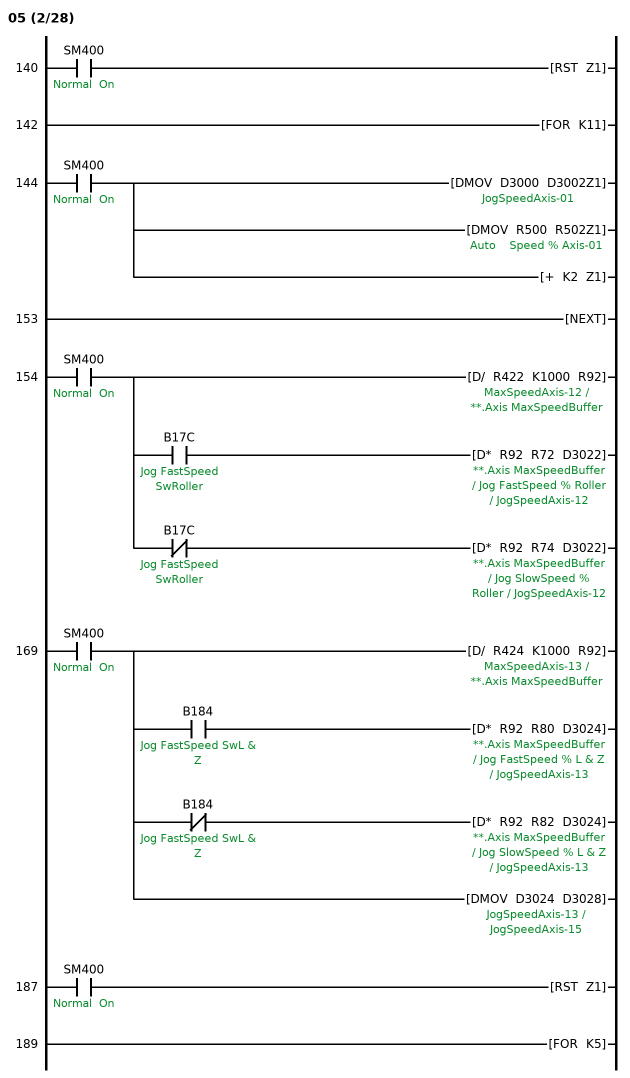
140   LD      SM400  ; Normal  On
      RST     Z1
142   FOR     K11
144   LD      SM400  ; Normal  On
      DMOV    D3000 D3002Z1
      DMOV    R500 R502Z1  ; Auto    Speed % Axis-01
      +       K2 Z1
153   NEXT
154   LD      SM400  ; Normal  On
      D/      R422 K1000 R92
      MPS
      AND     B17C  ; Jog FastSpeed SwRoller
      D*      R92 R72 D3022  ; Jog FastSpeed % Roller / JogSpeedAxis-12
      MPP
      ANI     B17C  ; Jog FastSpeed SwRoller
      D*      R92 R74 D3022  ; Jog SlowSpeed % Roller
169   LD      SM400  ; Normal  On
      D/      R424 K1000 R92
      MPS
      AND     B184  ; Jog FastSpeed SwL & Z
      D*      R92 R80 D3024  ; Jog FastSpeed % L & Z / JogSpeedAxis-13
      MRD
      ANI     B184  ; Jog FastSpeed SwL & Z
      D*      R92 R82 D3024  ; Jog SlowSpeed % L & Z
      MPP
      DMOV    D3024 D3028  ; JogSpeedAxis-15
187   LD      SM400  ; Normal  On
      RST     Z1
189   FOR     K5
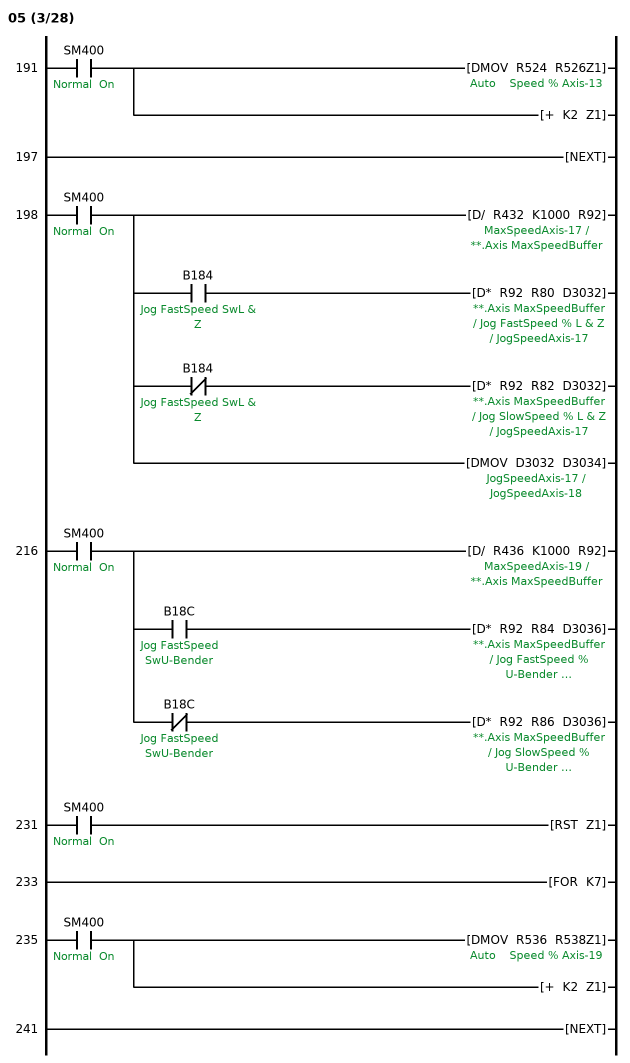
191   LD      SM400  ; Normal  On
      DMOV    R524 R526Z1  ; Auto    Speed % Axis-13
      +       K2 Z1
197   NEXT
198   LD      SM400  ; Normal  On
      D/      R432 K1000 R92  ; MaxSpeedAxis-17
      MPS
      AND     B184  ; Jog FastSpeed SwL & Z
      D*      R92 R80 D3032  ; JogSpeedAxis-17
      MRD
      ANI     B184  ; Jog FastSpeed SwL & Z
      D*      R92 R82 D3032
      MPP
      DMOV    D3032 D3034  ; JogSpeedAxis-18
216   LD      SM400  ; Normal  On
      D/      R436 K1000 R92
      MPS
      AND     B18C  ; Jog FastSpeed SwU-Bender
      D*      R92 R84 D3036  ; Jog FastSpeed % U-Bender / JogSpeedAxis-19
      MPP
      ANI     B18C  ; Jog FastSpeed SwU-Bender
      D*      R92 R86 D3036  ; Jog SlowSpeed % U-Bender
231   LD      SM400  ; Normal  On
      RST     Z1
233   FOR     K7
235   LD      SM400  ; Normal  On
      DMOV    R536 R538Z1  ; Auto    Speed % Axis-19
      +       K2 Z1
241   NEXT
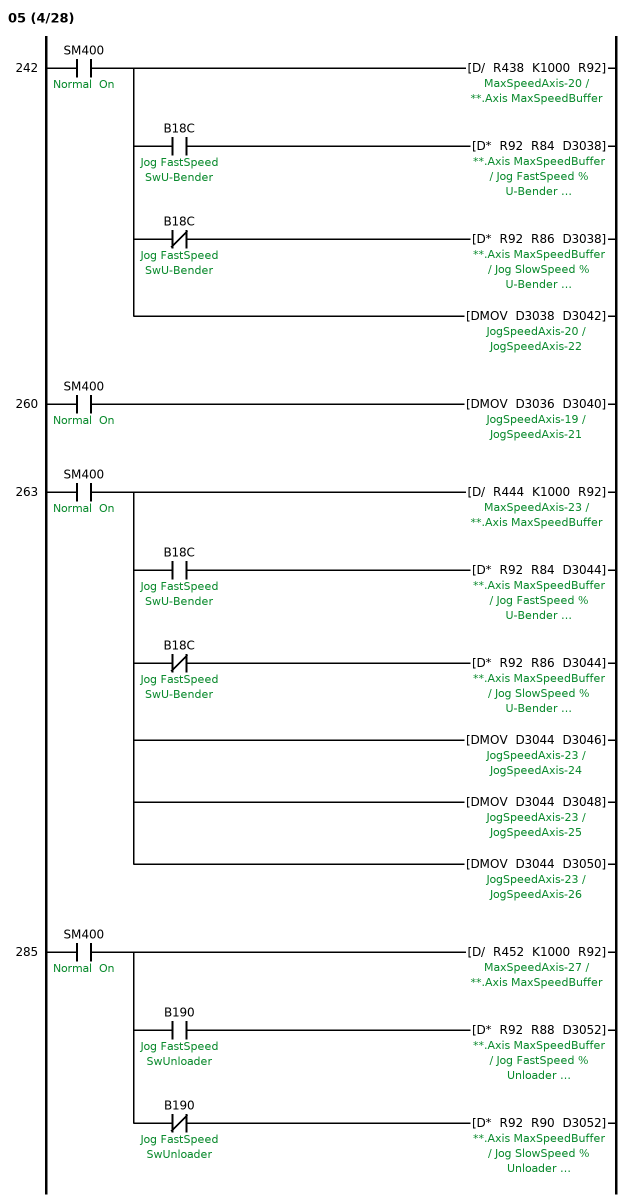
242   LD      SM400  ; Normal  On
      D/      R438 K1000 R92
      MPS
      AND     B18C  ; Jog FastSpeed SwU-Bender
      D*      R92 R84 D3038  ; JogSpeedAxis-20
      MRD
      ANI     B18C  ; Jog FastSpeed SwU-Bender
      D*      R92 R86 D3038
      MPP
      DMOV    D3038 D3042  ; JogSpeedAxis-22
260   LD      SM400  ; Normal  On
      DMOV    D3036 D3040  ; JogSpeedAxis-21
263   LD      SM400  ; Normal  On
      D/      R444 K1000 R92  ; MaxSpeedAxis-23
      MPS
      AND     B18C  ; Jog FastSpeed SwU-Bender
      D*      R92 R84 D3044  ; JogSpeedAxis-23
      MRD
      ANI     B18C  ; Jog FastSpeed SwU-Bender
      D*      R92 R86 D3044
      MPP
      DMOV    D3044 D3046  ; JogSpeedAxis-24
      DMOV    D3044 D3048  ; JogSpeedAxis-25
      DMOV    D3044 D3050  ; JogSpeedAxis-26
285   LD      SM400  ; Normal  On
      D/      R452 K1000 R92
      MPS
      AND     B190  ; Jog FastSpeed SwUnloader
      D*      R92 R88 D3052  ; Jog FastSpeed % Unloader / JogSpeedAxis-27
      MPP
      ANI     B190  ; Jog FastSpeed SwUnloader
      D*      R92 R90 D3052  ; Jog SlowSpeed % Unloader
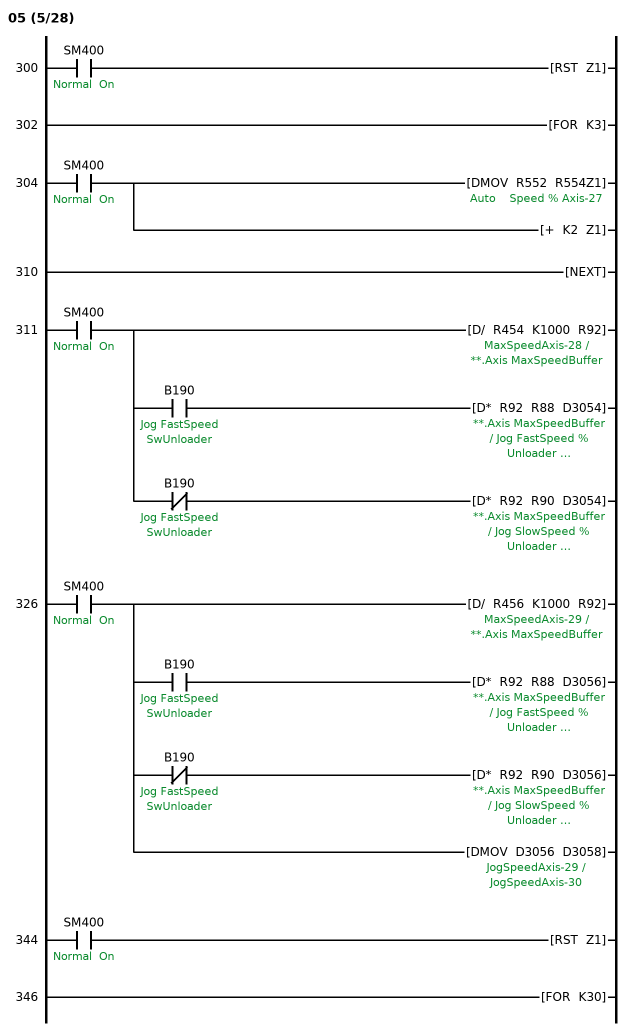
300   LD      SM400  ; Normal  On
      RST     Z1
302   FOR     K3
304   LD      SM400  ; Normal  On
      DMOV    R552 R554Z1  ; Auto    Speed % Axis-27
      +       K2 Z1
310   NEXT
311   LD      SM400  ; Normal  On
      D/      R454 K1000 R92
      MPS
      AND     B190  ; Jog FastSpeed SwUnloader
      D*      R92 R88 D3054  ; JogSpeedAxis-28
      MPP
      ANI     B190  ; Jog FastSpeed SwUnloader
      D*      R92 R90 D3054
326   LD      SM400  ; Normal  On
      D/      R456 K1000 R92  ; MaxSpeedAxis-29
      MPS
      AND     B190  ; Jog FastSpeed SwUnloader
      D*      R92 R88 D3056  ; JogSpeedAxis-29
      MRD
      ANI     B190  ; Jog FastSpeed SwUnloader
      D*      R92 R90 D3056
      MPP
      DMOV    D3056 D3058  ; JogSpeedAxis-30
344   LD      SM400  ; Normal  On
      RST     Z1
346   FOR     K30
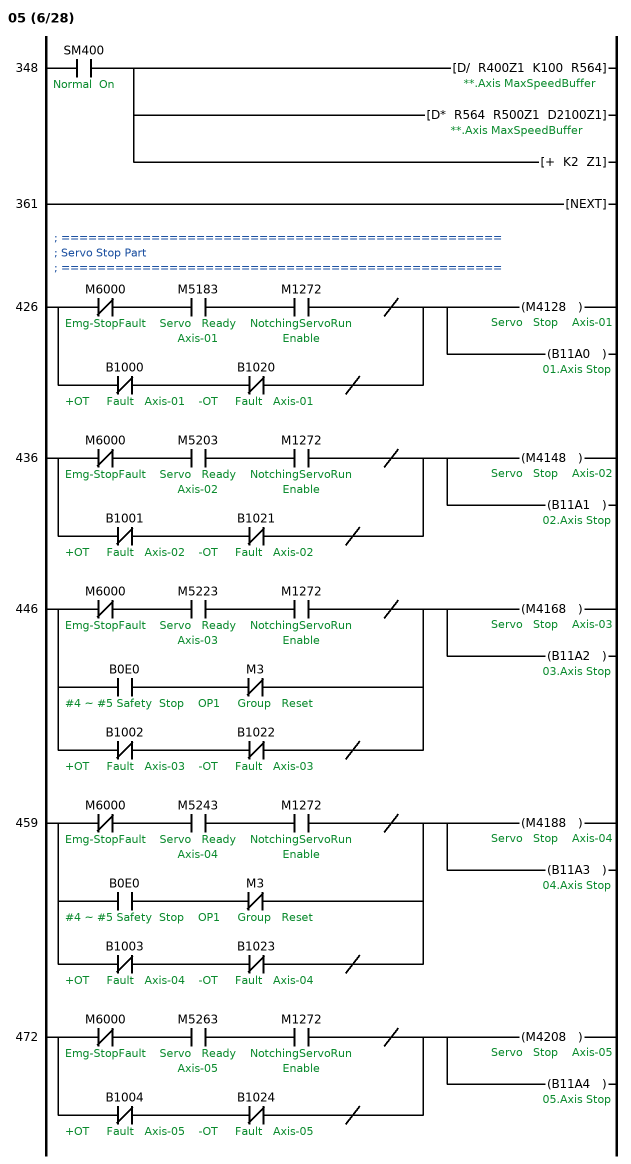
348   LD      SM400  ; Normal  On
      D/      R400Z1 K100 R564  ; **.Axis MaxSpeedBuffer
      D*      R564 R500Z1 D2100Z1
      +       K2 Z1
361   NEXT
; =================================================
; Servo Stop Part
; =================================================
426   LDI     M6000  ; Emg-StopFault
      AND     M5183  ; Servo   Ready   Axis-01
      AND     M1272  ; NotchingServoRunEnable
      INV
      LDI     B1000  ; +OT     Fault   Axis-01
      ANI     B1020  ; -OT     Fault   Axis-01
      INV
      ORB
      OUT     M4128  ; Servo   Stop    Axis-01
      OUT     B11A0  ; 01.Axis Stop
436   LDI     M6000  ; Emg-StopFault
      AND     M5203  ; Servo   Ready   Axis-02
      AND     M1272  ; NotchingServoRunEnable
      INV
      LDI     B1001  ; +OT     Fault   Axis-02
      ANI     B1021  ; -OT     Fault   Axis-02
      INV
      ORB
      OUT     M4148  ; Servo   Stop    Axis-02
      OUT     B11A1  ; 02.Axis Stop
446   LDI     M6000  ; Emg-StopFault
      AND     M5223  ; Servo   Ready   Axis-03
      AND     M1272  ; NotchingServoRunEnable
      INV
      LD      B0E0  ; #4 ~ #5 Safety  Stop
      ANI     M3  ; OP1     Group   Reset
      ORB
      LDI     B1002  ; +OT     Fault   Axis-03
      ANI     B1022  ; -OT     Fault   Axis-03
      INV
      ORB
      OUT     M4168  ; Servo   Stop    Axis-03
      OUT     B11A2  ; 03.Axis Stop
459   LDI     M6000  ; Emg-StopFault
      AND     M5243  ; Servo   Ready   Axis-04
      AND     M1272  ; NotchingServoRunEnable
      INV
      LD      B0E0  ; #4 ~ #5 Safety  Stop
      ANI     M3  ; OP1     Group   Reset
      ORB
      LDI     B1003  ; +OT     Fault   Axis-04
      ANI     B1023  ; -OT     Fault   Axis-04
      INV
      ORB
      OUT     M4188  ; Servo   Stop    Axis-04
      OUT     B11A3  ; 04.Axis Stop
472   LDI     M6000  ; Emg-StopFault
      AND     M5263  ; Servo   Ready   Axis-05
      AND     M1272  ; NotchingServoRunEnable
      INV
      LDI     B1004  ; +OT     Fault   Axis-05
      ANI     B1024  ; -OT     Fault   Axis-05
      INV
      ORB
      OUT     M4208  ; Servo   Stop    Axis-05
      OUT     B11A4  ; 05.Axis Stop
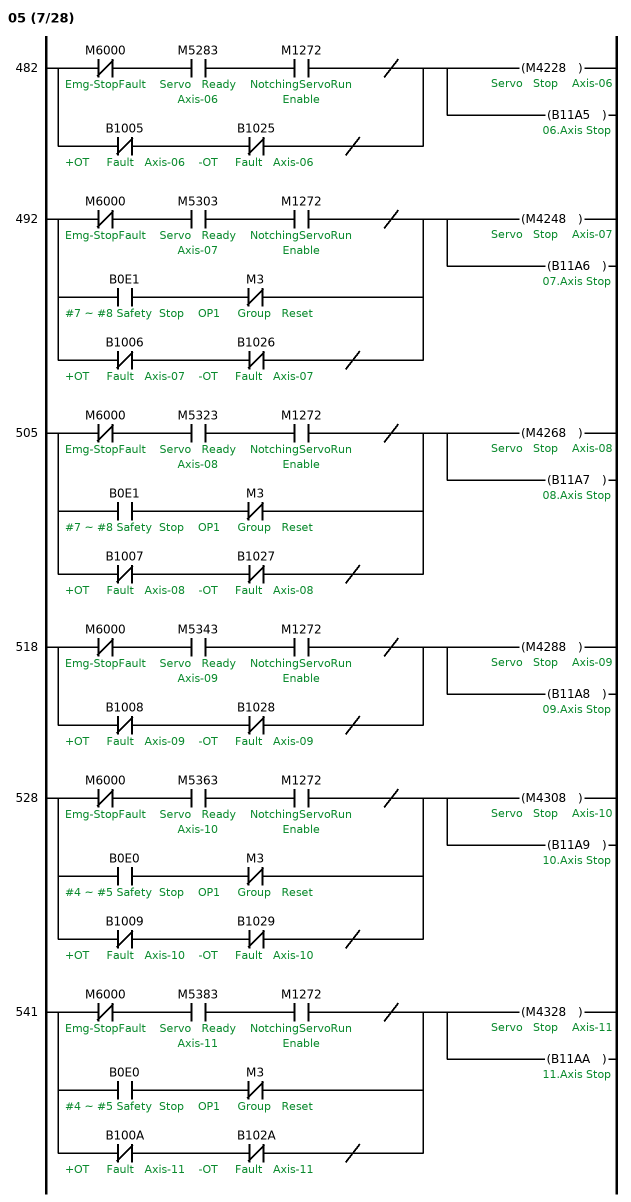
482   LDI     M6000  ; Emg-StopFault
      AND     M5283  ; Servo   Ready   Axis-06
      AND     M1272  ; NotchingServoRunEnable
      INV
      LDI     B1005  ; +OT     Fault   Axis-06
      ANI     B1025  ; -OT     Fault   Axis-06
      INV
      ORB
      OUT     M4228  ; Servo   Stop    Axis-06
      OUT     B11A5  ; 06.Axis Stop
492   LDI     M6000  ; Emg-StopFault
      AND     M5303  ; Servo   Ready   Axis-07
      AND     M1272  ; NotchingServoRunEnable
      INV
      LD      B0E1  ; #7 ~ #8 Safety  Stop
      ANI     M3  ; OP1     Group   Reset
      ORB
      LDI     B1006  ; +OT     Fault   Axis-07
      ANI     B1026  ; -OT     Fault   Axis-07
      INV
      ORB
      OUT     M4248  ; Servo   Stop    Axis-07
      OUT     B11A6  ; 07.Axis Stop
505   LDI     M6000  ; Emg-StopFault
      AND     M5323  ; Servo   Ready   Axis-08
      AND     M1272  ; NotchingServoRunEnable
      INV
      LD      B0E1  ; #7 ~ #8 Safety  Stop
      ANI     M3  ; OP1     Group   Reset
      ORB
      LDI     B1007  ; +OT     Fault   Axis-08
      ANI     B1027  ; -OT     Fault   Axis-08
      INV
      ORB
      OUT     M4268  ; Servo   Stop    Axis-08
      OUT     B11A7  ; 08.Axis Stop
518   LDI     M6000  ; Emg-StopFault
      AND     M5343  ; Servo   Ready   Axis-09
      AND     M1272  ; NotchingServoRunEnable
      INV
      LDI     B1008  ; +OT     Fault   Axis-09
      ANI     B1028  ; -OT     Fault   Axis-09
      INV
      ORB
      OUT     M4288  ; Servo   Stop    Axis-09
      OUT     B11A8  ; 09.Axis Stop
528   LDI     M6000  ; Emg-StopFault
      AND     M5363  ; Servo   Ready   Axis-10
      AND     M1272  ; NotchingServoRunEnable
      INV
      LD      B0E0  ; #4 ~ #5 Safety  Stop
      ANI     M3  ; OP1     Group   Reset
      ORB
      LDI     B1009  ; +OT     Fault   Axis-10
      ANI     B1029  ; -OT     Fault   Axis-10
      INV
      ORB
      OUT     M4308  ; Servo   Stop    Axis-10
      OUT     B11A9  ; 10.Axis Stop
541   LDI     M6000  ; Emg-StopFault
      AND     M5383  ; Servo   Ready   Axis-11
      AND     M1272  ; NotchingServoRunEnable
      INV
      LD      B0E0  ; #4 ~ #5 Safety  Stop
      ANI     M3  ; OP1     Group   Reset
      ORB
      LDI     B100A  ; +OT     Fault   Axis-11
      ANI     B102A  ; -OT     Fault   Axis-11
      INV
      ORB
      OUT     M4328  ; Servo   Stop    Axis-11
      OUT     B11AA  ; 11.Axis Stop
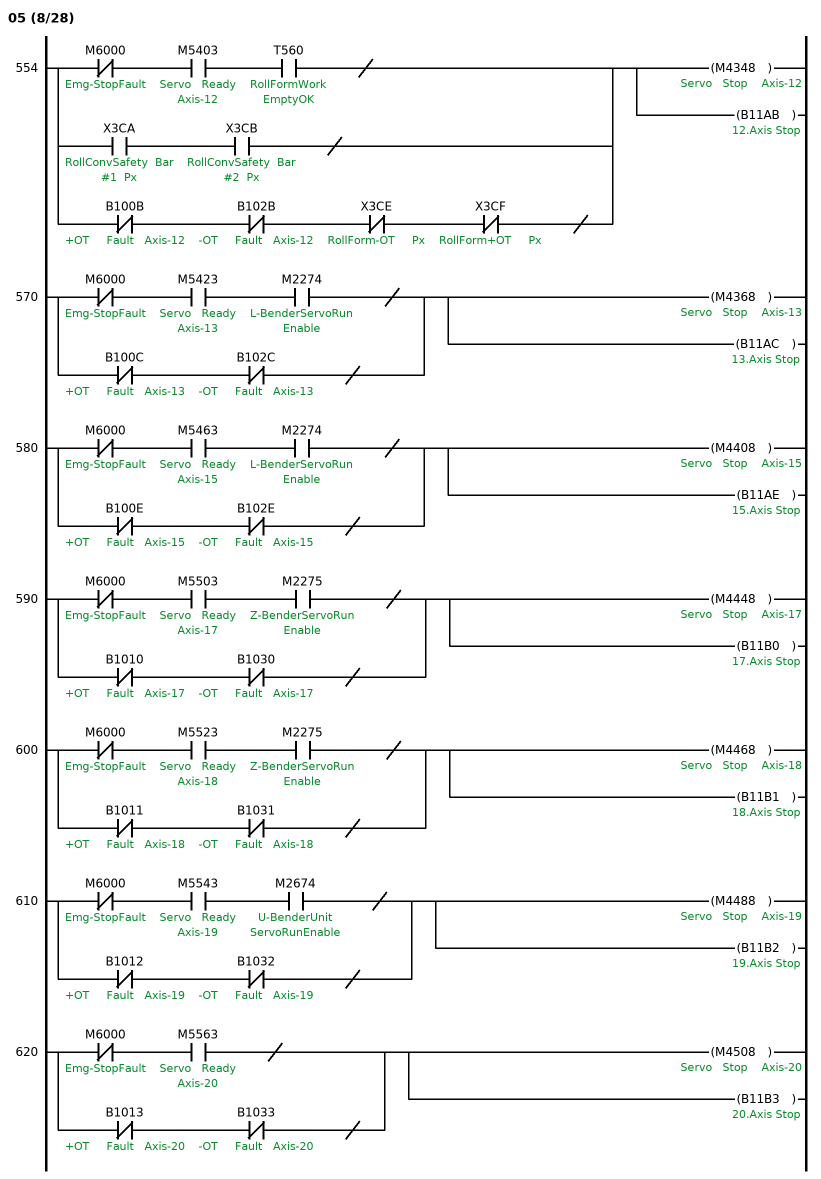
554   LDI     M6000  ; Emg-StopFault
      AND     M5403  ; Servo   Ready   Axis-12
      AND     T560  ; RollFormWork    EmptyOK
      INV
      LD      X3CA  ; RollConvSafety  Bar #1  Px
      AND     X3CB  ; RollConvSafety  Bar #2  Px
      INV
      ORB
      LDI     B100B  ; +OT     Fault   Axis-12
      ANI     B102B  ; -OT     Fault   Axis-12
      ANI     X3CE  ; RollForm-OT     Px
      ANI     X3CF  ; RollForm+OT     Px
      INV
      ORB
      OUT     M4348  ; Servo   Stop    Axis-12
      OUT     B11AB  ; 12.Axis Stop
570   LDI     M6000  ; Emg-StopFault
      AND     M5423  ; Servo   Ready   Axis-13
      AND     M2274  ; L-BenderServoRunEnable
      INV
      LDI     B100C  ; +OT     Fault   Axis-13
      ANI     B102C  ; -OT     Fault   Axis-13
      INV
      ORB
      OUT     M4368  ; Servo   Stop    Axis-13
      OUT     B11AC  ; 13.Axis Stop
580   LDI     M6000  ; Emg-StopFault
      AND     M5463  ; Servo   Ready   Axis-15
      AND     M2274  ; L-BenderServoRunEnable
      INV
      LDI     B100E  ; +OT     Fault   Axis-15
      ANI     B102E  ; -OT     Fault   Axis-15
      INV
      ORB
      OUT     M4408  ; Servo   Stop    Axis-15
      OUT     B11AE  ; 15.Axis Stop
590   LDI     M6000  ; Emg-StopFault
      AND     M5503  ; Servo   Ready   Axis-17
      AND     M2275  ; Z-BenderServoRunEnable
      INV
      LDI     B1010  ; +OT     Fault   Axis-17
      ANI     B1030  ; -OT     Fault   Axis-17
      INV
      ORB
      OUT     M4448  ; Servo   Stop    Axis-17
      OUT     B11B0  ; 17.Axis Stop
600   LDI     M6000  ; Emg-StopFault
      AND     M5523  ; Servo   Ready   Axis-18
      AND     M2275  ; Z-BenderServoRunEnable
      INV
      LDI     B1011  ; +OT     Fault   Axis-18
      ANI     B1031  ; -OT     Fault   Axis-18
      INV
      ORB
      OUT     M4468  ; Servo   Stop    Axis-18
      OUT     B11B1  ; 18.Axis Stop
610   LDI     M6000  ; Emg-StopFault
      AND     M5543  ; Servo   Ready   Axis-19
      AND     M2674  ; U-BenderUnit    ServoRunEnable
      INV
      LDI     B1012  ; +OT     Fault   Axis-19
      ANI     B1032  ; -OT     Fault   Axis-19
      INV
      ORB
      OUT     M4488  ; Servo   Stop    Axis-19
      OUT     B11B2  ; 19.Axis Stop
620   LDI     M6000  ; Emg-StopFault
      AND     M5563  ; Servo   Ready   Axis-20
      INV
      LDI     B1013  ; +OT     Fault   Axis-20
      ANI     B1033  ; -OT     Fault   Axis-20
      INV
      ORB
      OUT     M4508  ; Servo   Stop    Axis-20
      OUT     B11B3  ; 20.Axis Stop
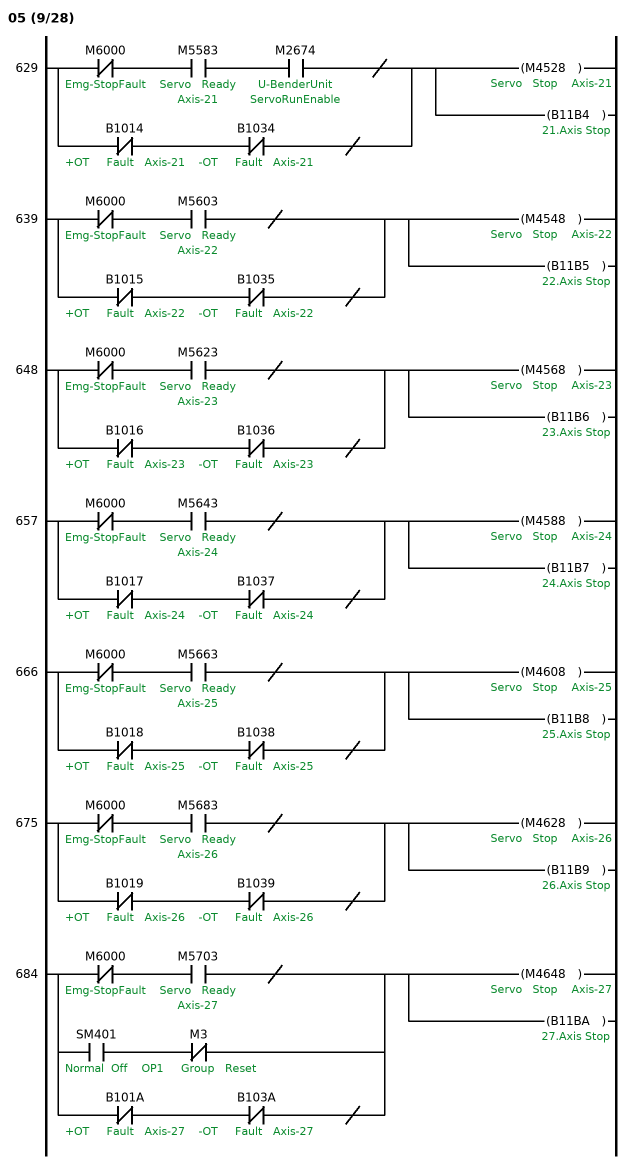
629   LDI     M6000  ; Emg-StopFault
      AND     M5583  ; Servo   Ready   Axis-21
      AND     M2674  ; U-BenderUnit    ServoRunEnable
      INV
      LDI     B1014  ; +OT     Fault   Axis-21
      ANI     B1034  ; -OT     Fault   Axis-21
      INV
      ORB
      OUT     M4528  ; Servo   Stop    Axis-21
      OUT     B11B4  ; 21.Axis Stop
639   LDI     M6000  ; Emg-StopFault
      AND     M5603  ; Servo   Ready   Axis-22
      INV
      LDI     B1015  ; +OT     Fault   Axis-22
      ANI     B1035  ; -OT     Fault   Axis-22
      INV
      ORB
      OUT     M4548  ; Servo   Stop    Axis-22
      OUT     B11B5  ; 22.Axis Stop
648   LDI     M6000  ; Emg-StopFault
      AND     M5623  ; Servo   Ready   Axis-23
      INV
      LDI     B1016  ; +OT     Fault   Axis-23
      ANI     B1036  ; -OT     Fault   Axis-23
      INV
      ORB
      OUT     M4568  ; Servo   Stop    Axis-23
      OUT     B11B6  ; 23.Axis Stop
657   LDI     M6000  ; Emg-StopFault
      AND     M5643  ; Servo   Ready   Axis-24
      INV
      LDI     B1017  ; +OT     Fault   Axis-24
      ANI     B1037  ; -OT     Fault   Axis-24
      INV
      ORB
      OUT     M4588  ; Servo   Stop    Axis-24
      OUT     B11B7  ; 24.Axis Stop
666   LDI     M6000  ; Emg-StopFault
      AND     M5663  ; Servo   Ready   Axis-25
      INV
      LDI     B1018  ; +OT     Fault   Axis-25
      ANI     B1038  ; -OT     Fault   Axis-25
      INV
      ORB
      OUT     M4608  ; Servo   Stop    Axis-25
      OUT     B11B8  ; 25.Axis Stop
675   LDI     M6000  ; Emg-StopFault
      AND     M5683  ; Servo   Ready   Axis-26
      INV
      LDI     B1019  ; +OT     Fault   Axis-26
      ANI     B1039  ; -OT     Fault   Axis-26
      INV
      ORB
      OUT     M4628  ; Servo   Stop    Axis-26
      OUT     B11B9  ; 26.Axis Stop
684   LDI     M6000  ; Emg-StopFault
      AND     M5703  ; Servo   Ready   Axis-27
      INV
      LD      SM401  ; Normal  Off
      ANI     M3  ; OP1     Group   Reset
      ORB
      LDI     B101A  ; +OT     Fault   Axis-27
      ANI     B103A  ; -OT     Fault   Axis-27
      INV
      ORB
      OUT     M4648  ; Servo   Stop    Axis-27
      OUT     B11BA  ; 27.Axis Stop
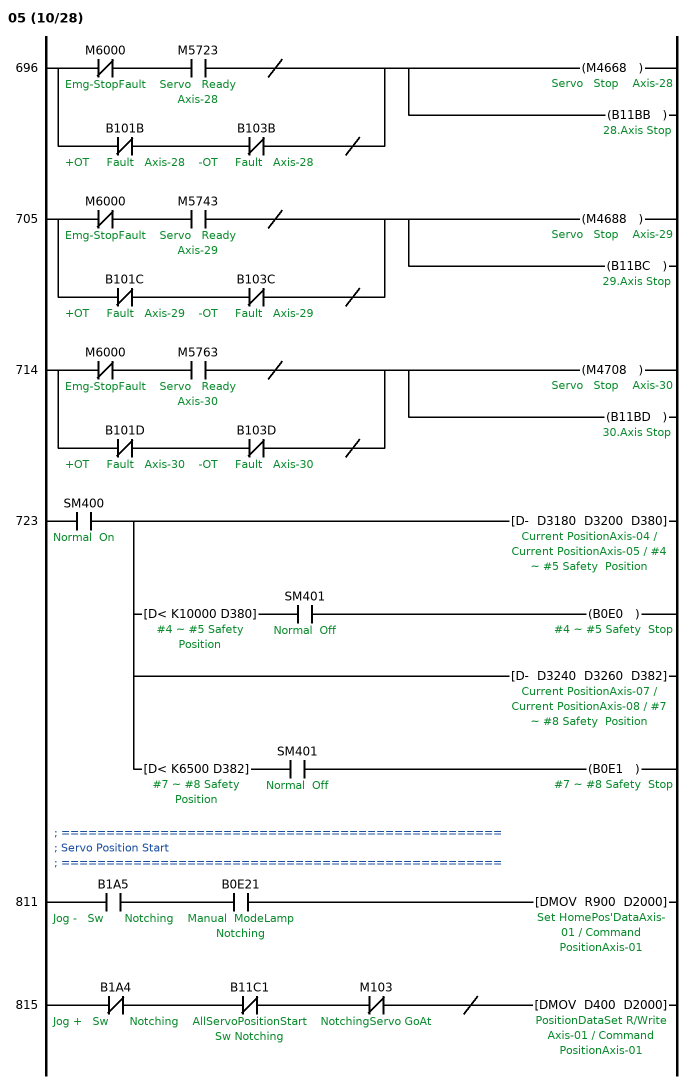
696   LDI     M6000  ; Emg-StopFault
      AND     M5723  ; Servo   Ready   Axis-28
      INV
      LDI     B101B  ; +OT     Fault   Axis-28
      ANI     B103B  ; -OT     Fault   Axis-28
      INV
      ORB
      OUT     M4668  ; Servo   Stop    Axis-28
      OUT     B11BB  ; 28.Axis Stop
705   LDI     M6000  ; Emg-StopFault
      AND     M5743  ; Servo   Ready   Axis-29
      INV
      LDI     B101C  ; +OT     Fault   Axis-29
      ANI     B103C  ; -OT     Fault   Axis-29
      INV
      ORB
      OUT     M4688  ; Servo   Stop    Axis-29
      OUT     B11BC  ; 29.Axis Stop
714   LDI     M6000  ; Emg-StopFault
      AND     M5763  ; Servo   Ready   Axis-30
      INV
      LDI     B101D  ; +OT     Fault   Axis-30
      ANI     B103D  ; -OT     Fault   Axis-30
      INV
      ORB
      OUT     M4708  ; Servo   Stop    Axis-30
      OUT     B11BD  ; 30.Axis Stop
723   LD      SM400  ; Normal  On
      D-      D3180 D3200 D380  ; Current PositionAxis-04 / Current PositionAxis-05 / #4 ~ #5 Safety  Position
      MPS
      ANDD<   K10000 D380  ; #4 ~ #5 Safety  Position
      AND     SM401  ; Normal  Off
      OUT     B0E0  ; #4 ~ #5 Safety  Stop
      MPP
      D-      D3240 D3260 D382  ; Current PositionAxis-07 / Current PositionAxis-08 / #7 ~ #8 Safety  Position
      ANDD<   K6500 D382  ; #7 ~ #8 Safety  Position
      AND     SM401  ; Normal  Off
      OUT     B0E1  ; #7 ~ #8 Safety  Stop
; =================================================
; Servo Position Start
; =================================================
811   LD      B1A5  ; Jog -   Sw      Notching
      AND     B0E21  ; Manual  ModeLampNotching
      DMOV    R900 D2000  ; Set HomePos'DataAxis-01 / Command PositionAxis-01
815   LDI     B1A4  ; Jog +   Sw      Notching
      ANI     B11C1  ; AllServoPositionStartSw Notching
      ANI     M103  ; NotchingServo GoAt
      INV
      DMOV    D400 D2000  ; PositionDataSet R/Write Axis-01
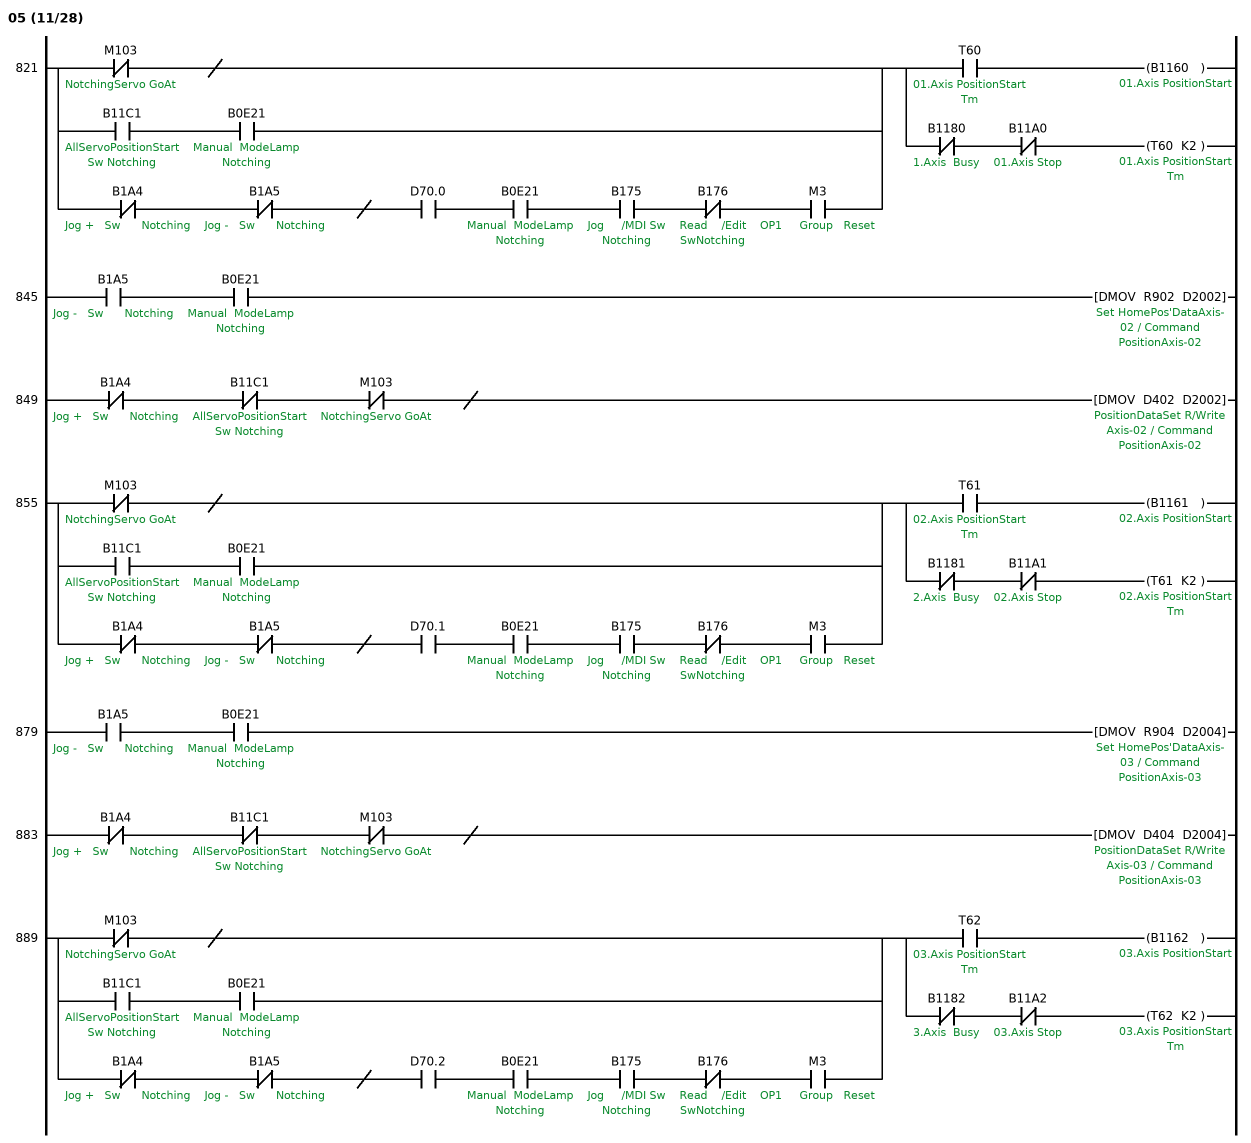
821   LDI     M103  ; NotchingServo GoAt
      INV
      LD      B11C1  ; AllServoPositionStartSw Notching
      AND     B0E21  ; Manual  ModeLampNotching
      ORB
      LDI     B1A4  ; Jog +   Sw      Notching
      ANI     B1A5  ; Jog -   Sw      Notching
      INV
      AND     D70.0
      AND     B0E21  ; Manual  ModeLampNotching
      AND     B175  ; Jog     /MDI Sw Notching
      ANI     B176  ; Read    /Edit SwNotching
      AND     M3  ; OP1     Group   Reset
      ORB
      MPS
      AND     T60  ; 01.Axis PositionStart Tm
      OUT     B1160  ; 01.Axis PositionStart
      MPP
      ANI     B1180  ; 1.Axis  Busy
      ANI     B11A0  ; 01.Axis Stop
      OUT     T60 K2  ; 01.Axis PositionStart Tm
845   LD      B1A5  ; Jog -   Sw      Notching
      AND     B0E21  ; Manual  ModeLampNotching
      DMOV    R902 D2002  ; Set HomePos'DataAxis-02 / Command PositionAxis-02
849   LDI     B1A4  ; Jog +   Sw      Notching
      ANI     B11C1  ; AllServoPositionStartSw Notching
      ANI     M103  ; NotchingServo GoAt
      INV
      DMOV    D402 D2002  ; PositionDataSet R/Write Axis-02
855   LDI     M103  ; NotchingServo GoAt
      INV
      LD      B11C1  ; AllServoPositionStartSw Notching
      AND     B0E21  ; Manual  ModeLampNotching
      ORB
      LDI     B1A4  ; Jog +   Sw      Notching
      ANI     B1A5  ; Jog -   Sw      Notching
      INV
      AND     D70.1
      AND     B0E21  ; Manual  ModeLampNotching
      AND     B175  ; Jog     /MDI Sw Notching
      ANI     B176  ; Read    /Edit SwNotching
      AND     M3  ; OP1     Group   Reset
      ORB
      MPS
      AND     T61  ; 02.Axis PositionStart Tm
      OUT     B1161  ; 02.Axis PositionStart
      MPP
      ANI     B1181  ; 2.Axis  Busy
      ANI     B11A1  ; 02.Axis Stop
      OUT     T61 K2  ; 02.Axis PositionStart Tm
879   LD      B1A5  ; Jog -   Sw      Notching
      AND     B0E21  ; Manual  ModeLampNotching
      DMOV    R904 D2004  ; Set HomePos'DataAxis-03 / Command PositionAxis-03
883   LDI     B1A4  ; Jog +   Sw      Notching
      ANI     B11C1  ; AllServoPositionStartSw Notching
      ANI     M103  ; NotchingServo GoAt
      INV
      DMOV    D404 D2004  ; PositionDataSet R/Write Axis-03
889   LDI     M103  ; NotchingServo GoAt
      INV
      LD      B11C1  ; AllServoPositionStartSw Notching
      AND     B0E21  ; Manual  ModeLampNotching
      ORB
      LDI     B1A4  ; Jog +   Sw      Notching
      ANI     B1A5  ; Jog -   Sw      Notching
      INV
      AND     D70.2
      AND     B0E21  ; Manual  ModeLampNotching
      AND     B175  ; Jog     /MDI Sw Notching
      ANI     B176  ; Read    /Edit SwNotching
      AND     M3  ; OP1     Group   Reset
      ORB
      MPS
      AND     T62  ; 03.Axis PositionStart Tm
      OUT     B1162  ; 03.Axis PositionStart
      MPP
      ANI     B1182  ; 3.Axis  Busy
      ANI     B11A2  ; 03.Axis Stop
      OUT     T62 K2  ; 03.Axis PositionStart Tm
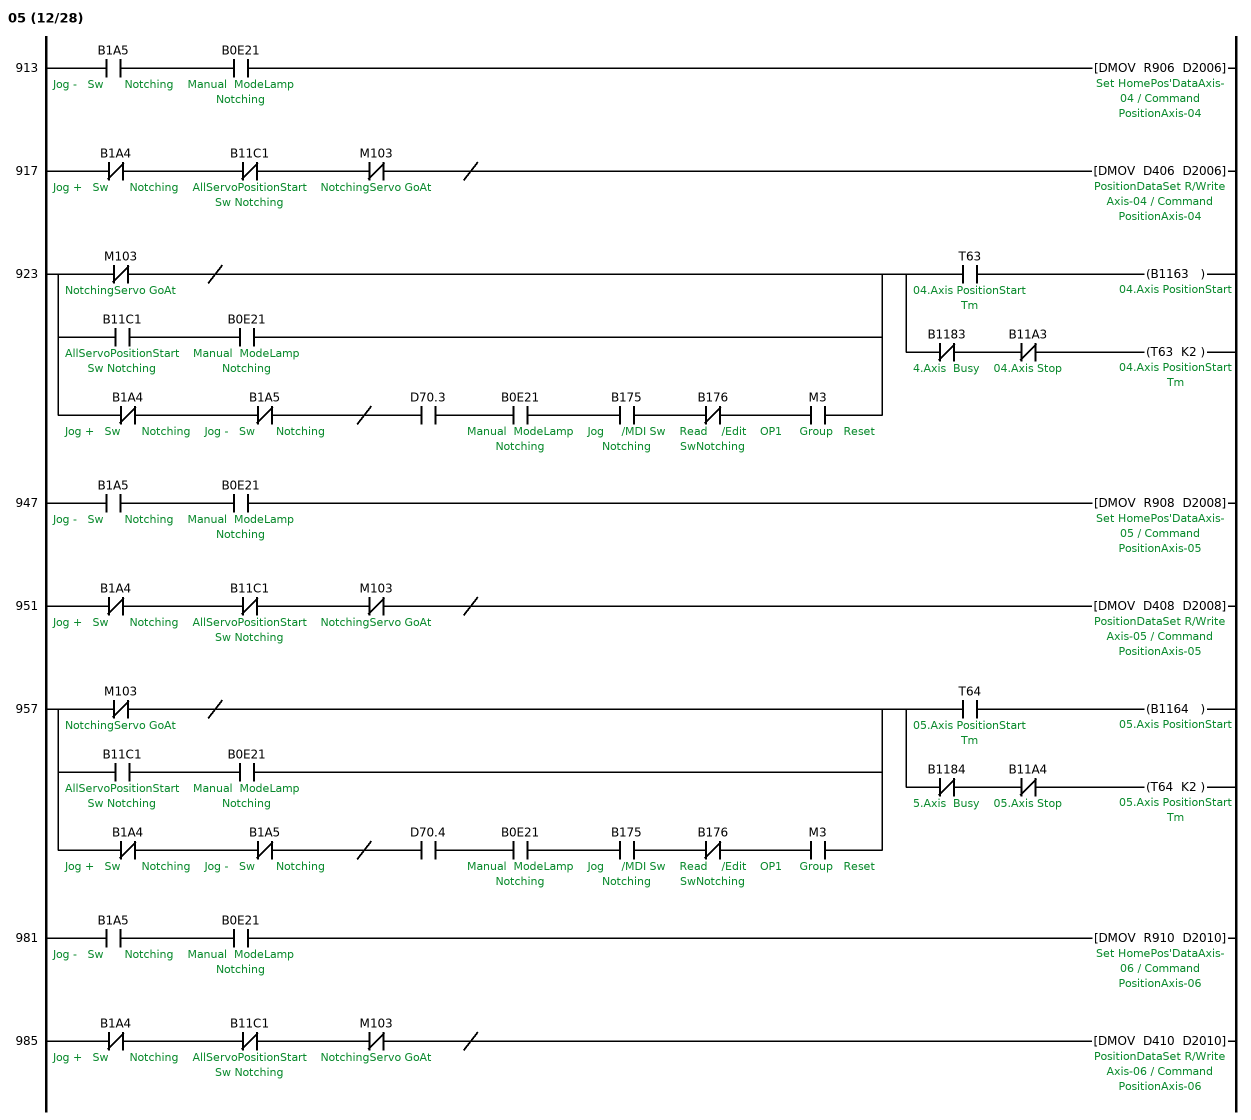
913   LD      B1A5  ; Jog -   Sw      Notching
      AND     B0E21  ; Manual  ModeLampNotching
      DMOV    R906 D2006  ; Set HomePos'DataAxis-04 / Command PositionAxis-04
917   LDI     B1A4  ; Jog +   Sw      Notching
      ANI     B11C1  ; AllServoPositionStartSw Notching
      ANI     M103  ; NotchingServo GoAt
      INV
      DMOV    D406 D2006  ; PositionDataSet R/Write Axis-04
923   LDI     M103  ; NotchingServo GoAt
      INV
      LD      B11C1  ; AllServoPositionStartSw Notching
      AND     B0E21  ; Manual  ModeLampNotching
      ORB
      LDI     B1A4  ; Jog +   Sw      Notching
      ANI     B1A5  ; Jog -   Sw      Notching
      INV
      AND     D70.3
      AND     B0E21  ; Manual  ModeLampNotching
      AND     B175  ; Jog     /MDI Sw Notching
      ANI     B176  ; Read    /Edit SwNotching
      AND     M3  ; OP1     Group   Reset
      ORB
      MPS
      AND     T63  ; 04.Axis PositionStart Tm
      OUT     B1163  ; 04.Axis PositionStart
      MPP
      ANI     B1183  ; 4.Axis  Busy
      ANI     B11A3  ; 04.Axis Stop
      OUT     T63 K2  ; 04.Axis PositionStart Tm
947   LD      B1A5  ; Jog -   Sw      Notching
      AND     B0E21  ; Manual  ModeLampNotching
      DMOV    R908 D2008  ; Set HomePos'DataAxis-05 / Command PositionAxis-05
951   LDI     B1A4  ; Jog +   Sw      Notching
      ANI     B11C1  ; AllServoPositionStartSw Notching
      ANI     M103  ; NotchingServo GoAt
      INV
      DMOV    D408 D2008  ; PositionDataSet R/Write Axis-05
957   LDI     M103  ; NotchingServo GoAt
      INV
      LD      B11C1  ; AllServoPositionStartSw Notching
      AND     B0E21  ; Manual  ModeLampNotching
      ORB
      LDI     B1A4  ; Jog +   Sw      Notching
      ANI     B1A5  ; Jog -   Sw      Notching
      INV
      AND     D70.4
      AND     B0E21  ; Manual  ModeLampNotching
      AND     B175  ; Jog     /MDI Sw Notching
      ANI     B176  ; Read    /Edit SwNotching
      AND     M3  ; OP1     Group   Reset
      ORB
      MPS
      AND     T64  ; 05.Axis PositionStart Tm
      OUT     B1164  ; 05.Axis PositionStart
      MPP
      ANI     B1184  ; 5.Axis  Busy
      ANI     B11A4  ; 05.Axis Stop
      OUT     T64 K2  ; 05.Axis PositionStart Tm
981   LD      B1A5  ; Jog -   Sw      Notching
      AND     B0E21  ; Manual  ModeLampNotching
      DMOV    R910 D2010  ; Set HomePos'DataAxis-06 / Command PositionAxis-06
985   LDI     B1A4  ; Jog +   Sw      Notching
      ANI     B11C1  ; AllServoPositionStartSw Notching
      ANI     M103  ; NotchingServo GoAt
      INV
      DMOV    D410 D2010  ; PositionDataSet R/Write Axis-06
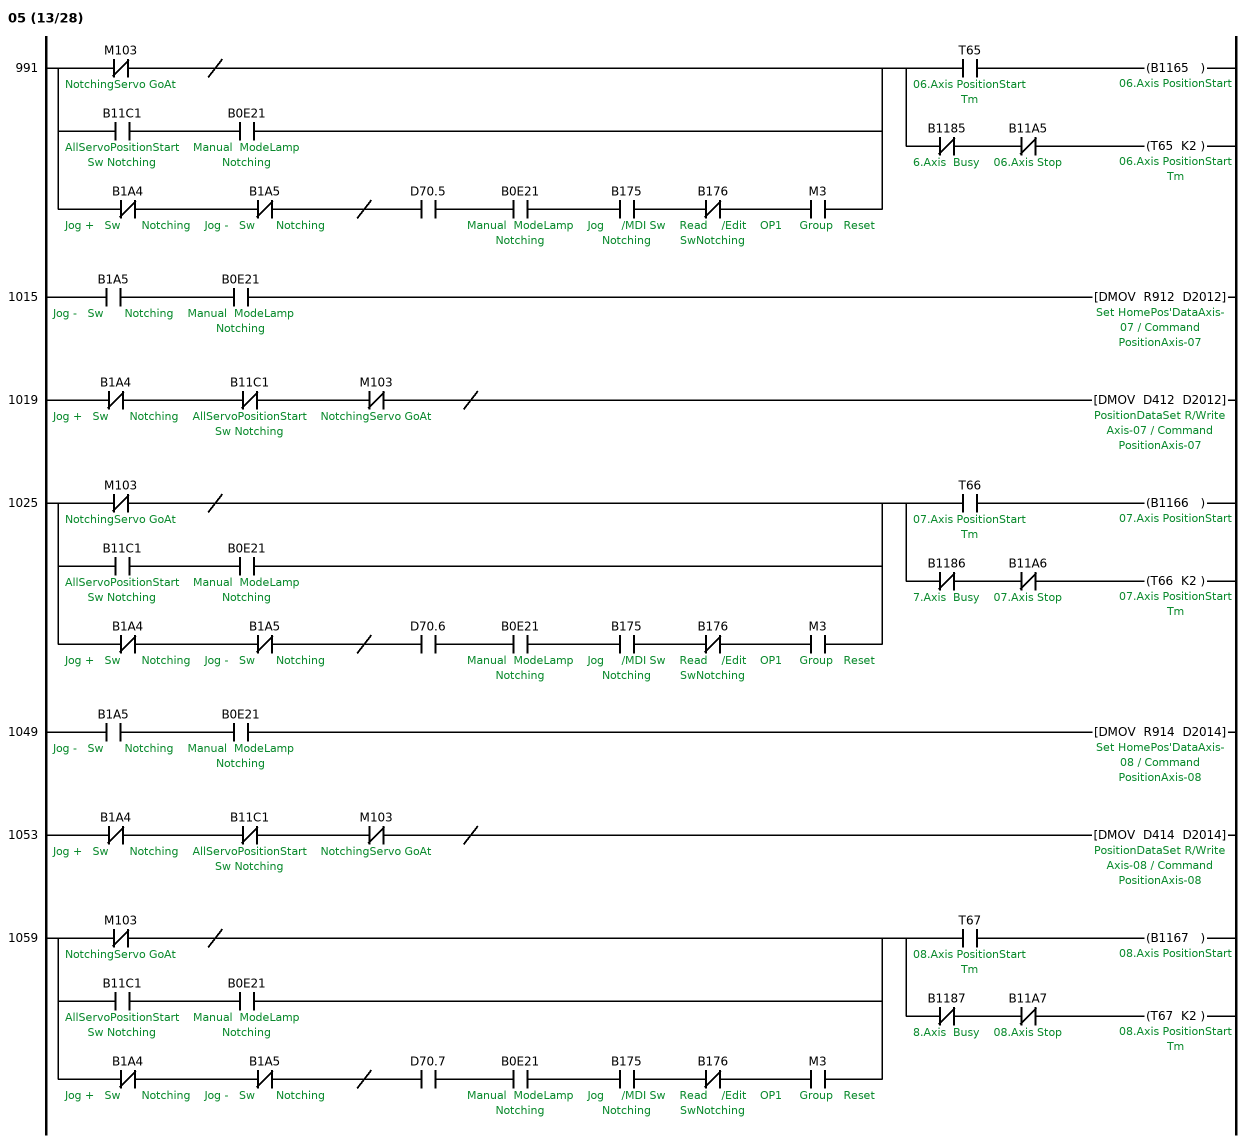
991   LDI     M103  ; NotchingServo GoAt
      INV
      LD      B11C1  ; AllServoPositionStartSw Notching
      AND     B0E21  ; Manual  ModeLampNotching
      ORB
      LDI     B1A4  ; Jog +   Sw      Notching
      ANI     B1A5  ; Jog -   Sw      Notching
      INV
      AND     D70.5
      AND     B0E21  ; Manual  ModeLampNotching
      AND     B175  ; Jog     /MDI Sw Notching
      ANI     B176  ; Read    /Edit SwNotching
      AND     M3  ; OP1     Group   Reset
      ORB
      MPS
      AND     T65  ; 06.Axis PositionStart Tm
      OUT     B1165  ; 06.Axis PositionStart
      MPP
      ANI     B1185  ; 6.Axis  Busy
      ANI     B11A5  ; 06.Axis Stop
      OUT     T65 K2  ; 06.Axis PositionStart Tm
1015  LD      B1A5  ; Jog -   Sw      Notching
      AND     B0E21  ; Manual  ModeLampNotching
      DMOV    R912 D2012  ; Set HomePos'DataAxis-07 / Command PositionAxis-07
1019  LDI     B1A4  ; Jog +   Sw      Notching
      ANI     B11C1  ; AllServoPositionStartSw Notching
      ANI     M103  ; NotchingServo GoAt
      INV
      DMOV    D412 D2012  ; PositionDataSet R/Write Axis-07
1025  LDI     M103  ; NotchingServo GoAt
      INV
      LD      B11C1  ; AllServoPositionStartSw Notching
      AND     B0E21  ; Manual  ModeLampNotching
      ORB
      LDI     B1A4  ; Jog +   Sw      Notching
      ANI     B1A5  ; Jog -   Sw      Notching
      INV
      AND     D70.6
      AND     B0E21  ; Manual  ModeLampNotching
      AND     B175  ; Jog     /MDI Sw Notching
      ANI     B176  ; Read    /Edit SwNotching
      AND     M3  ; OP1     Group   Reset
      ORB
      MPS
      AND     T66  ; 07.Axis PositionStart Tm
      OUT     B1166  ; 07.Axis PositionStart
      MPP
      ANI     B1186  ; 7.Axis  Busy
      ANI     B11A6  ; 07.Axis Stop
      OUT     T66 K2  ; 07.Axis PositionStart Tm
1049  LD      B1A5  ; Jog -   Sw      Notching
      AND     B0E21  ; Manual  ModeLampNotching
      DMOV    R914 D2014  ; Set HomePos'DataAxis-08 / Command PositionAxis-08
1053  LDI     B1A4  ; Jog +   Sw      Notching
      ANI     B11C1  ; AllServoPositionStartSw Notching
      ANI     M103  ; NotchingServo GoAt
      INV
      DMOV    D414 D2014  ; PositionDataSet R/Write Axis-08
1059  LDI     M103  ; NotchingServo GoAt
      INV
      LD      B11C1  ; AllServoPositionStartSw Notching
      AND     B0E21  ; Manual  ModeLampNotching
      ORB
      LDI     B1A4  ; Jog +   Sw      Notching
      ANI     B1A5  ; Jog -   Sw      Notching
      INV
      AND     D70.7
      AND     B0E21  ; Manual  ModeLampNotching
      AND     B175  ; Jog     /MDI Sw Notching
      ANI     B176  ; Read    /Edit SwNotching
      AND     M3  ; OP1     Group   Reset
      ORB
      MPS
      AND     T67  ; 08.Axis PositionStart Tm
      OUT     B1167  ; 08.Axis PositionStart
      MPP
      ANI     B1187  ; 8.Axis  Busy
      ANI     B11A7  ; 08.Axis Stop
      OUT     T67 K2  ; 08.Axis PositionStart Tm
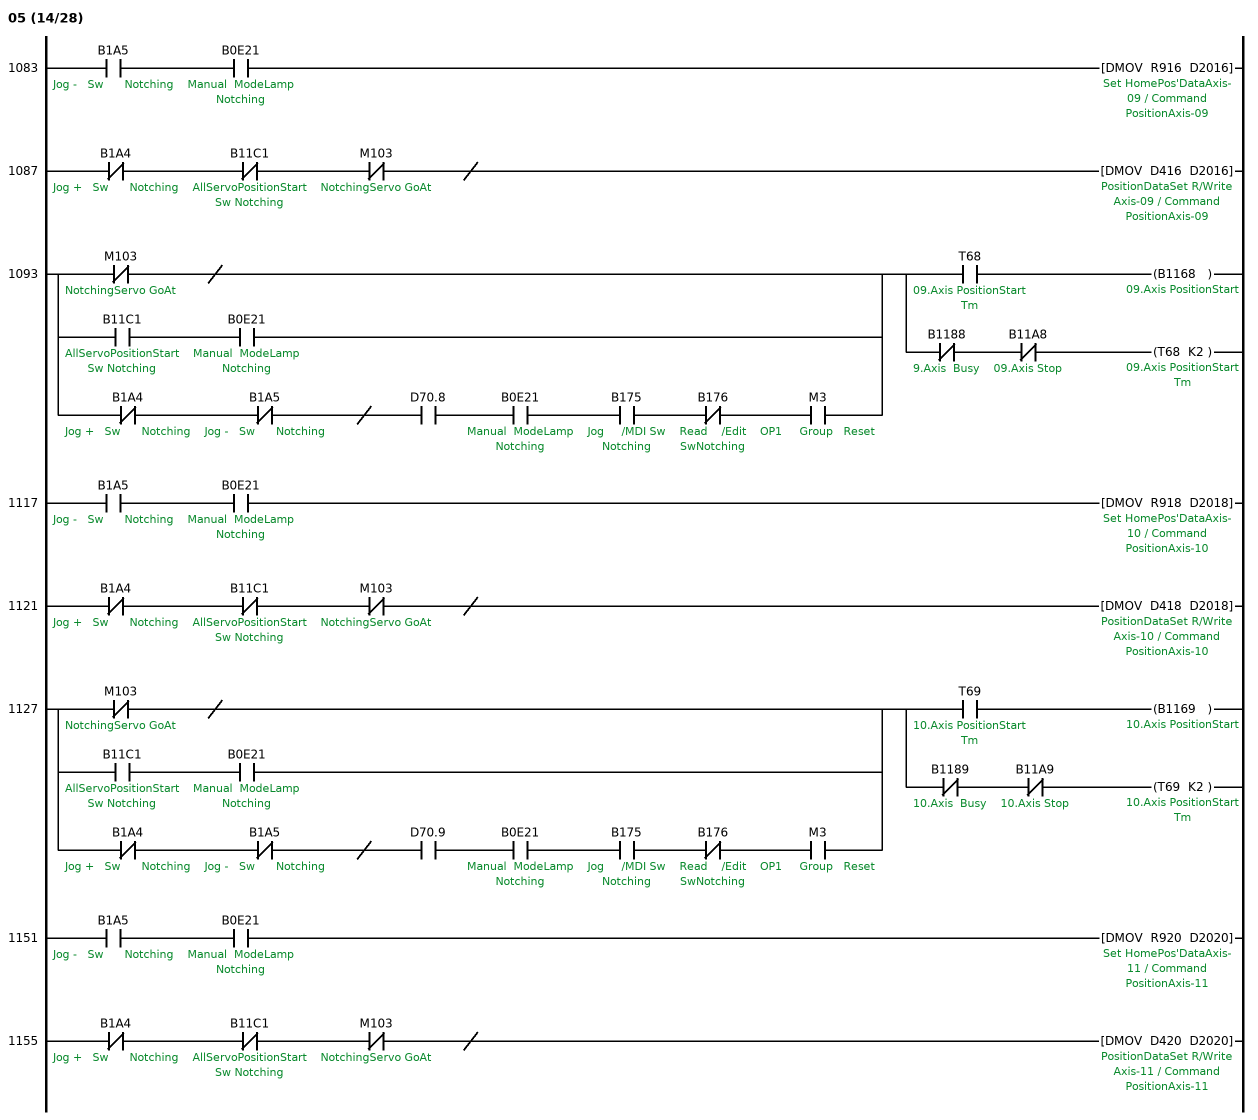
1083  LD      B1A5  ; Jog -   Sw      Notching
      AND     B0E21  ; Manual  ModeLampNotching
      DMOV    R916 D2016  ; Set HomePos'DataAxis-09 / Command PositionAxis-09
1087  LDI     B1A4  ; Jog +   Sw      Notching
      ANI     B11C1  ; AllServoPositionStartSw Notching
      ANI     M103  ; NotchingServo GoAt
      INV
      DMOV    D416 D2016  ; PositionDataSet R/Write Axis-09
1093  LDI     M103  ; NotchingServo GoAt
      INV
      LD      B11C1  ; AllServoPositionStartSw Notching
      AND     B0E21  ; Manual  ModeLampNotching
      ORB
      LDI     B1A4  ; Jog +   Sw      Notching
      ANI     B1A5  ; Jog -   Sw      Notching
      INV
      AND     D70.8
      AND     B0E21  ; Manual  ModeLampNotching
      AND     B175  ; Jog     /MDI Sw Notching
      ANI     B176  ; Read    /Edit SwNotching
      AND     M3  ; OP1     Group   Reset
      ORB
      MPS
      AND     T68  ; 09.Axis PositionStart Tm
      OUT     B1168  ; 09.Axis PositionStart
      MPP
      ANI     B1188  ; 9.Axis  Busy
      ANI     B11A8  ; 09.Axis Stop
      OUT     T68 K2  ; 09.Axis PositionStart Tm
1117  LD      B1A5  ; Jog -   Sw      Notching
      AND     B0E21  ; Manual  ModeLampNotching
      DMOV    R918 D2018  ; Set HomePos'DataAxis-10 / Command PositionAxis-10
1121  LDI     B1A4  ; Jog +   Sw      Notching
      ANI     B11C1  ; AllServoPositionStartSw Notching
      ANI     M103  ; NotchingServo GoAt
      INV
      DMOV    D418 D2018  ; PositionDataSet R/Write Axis-10
1127  LDI     M103  ; NotchingServo GoAt
      INV
      LD      B11C1  ; AllServoPositionStartSw Notching
      AND     B0E21  ; Manual  ModeLampNotching
      ORB
      LDI     B1A4  ; Jog +   Sw      Notching
      ANI     B1A5  ; Jog -   Sw      Notching
      INV
      AND     D70.9
      AND     B0E21  ; Manual  ModeLampNotching
      AND     B175  ; Jog     /MDI Sw Notching
      ANI     B176  ; Read    /Edit SwNotching
      AND     M3  ; OP1     Group   Reset
      ORB
      MPS
      AND     T69  ; 10.Axis PositionStart Tm
      OUT     B1169  ; 10.Axis PositionStart
      MPP
      ANI     B1189  ; 10.Axis  Busy
      ANI     B11A9  ; 10.Axis Stop
      OUT     T69 K2  ; 10.Axis PositionStart Tm
1151  LD      B1A5  ; Jog -   Sw      Notching
      AND     B0E21  ; Manual  ModeLampNotching
      DMOV    R920 D2020  ; Set HomePos'DataAxis-11 / Command PositionAxis-11
1155  LDI     B1A4  ; Jog +   Sw      Notching
      ANI     B11C1  ; AllServoPositionStartSw Notching
      ANI     M103  ; NotchingServo GoAt
      INV
      DMOV    D420 D2020  ; PositionDataSet R/Write Axis-11
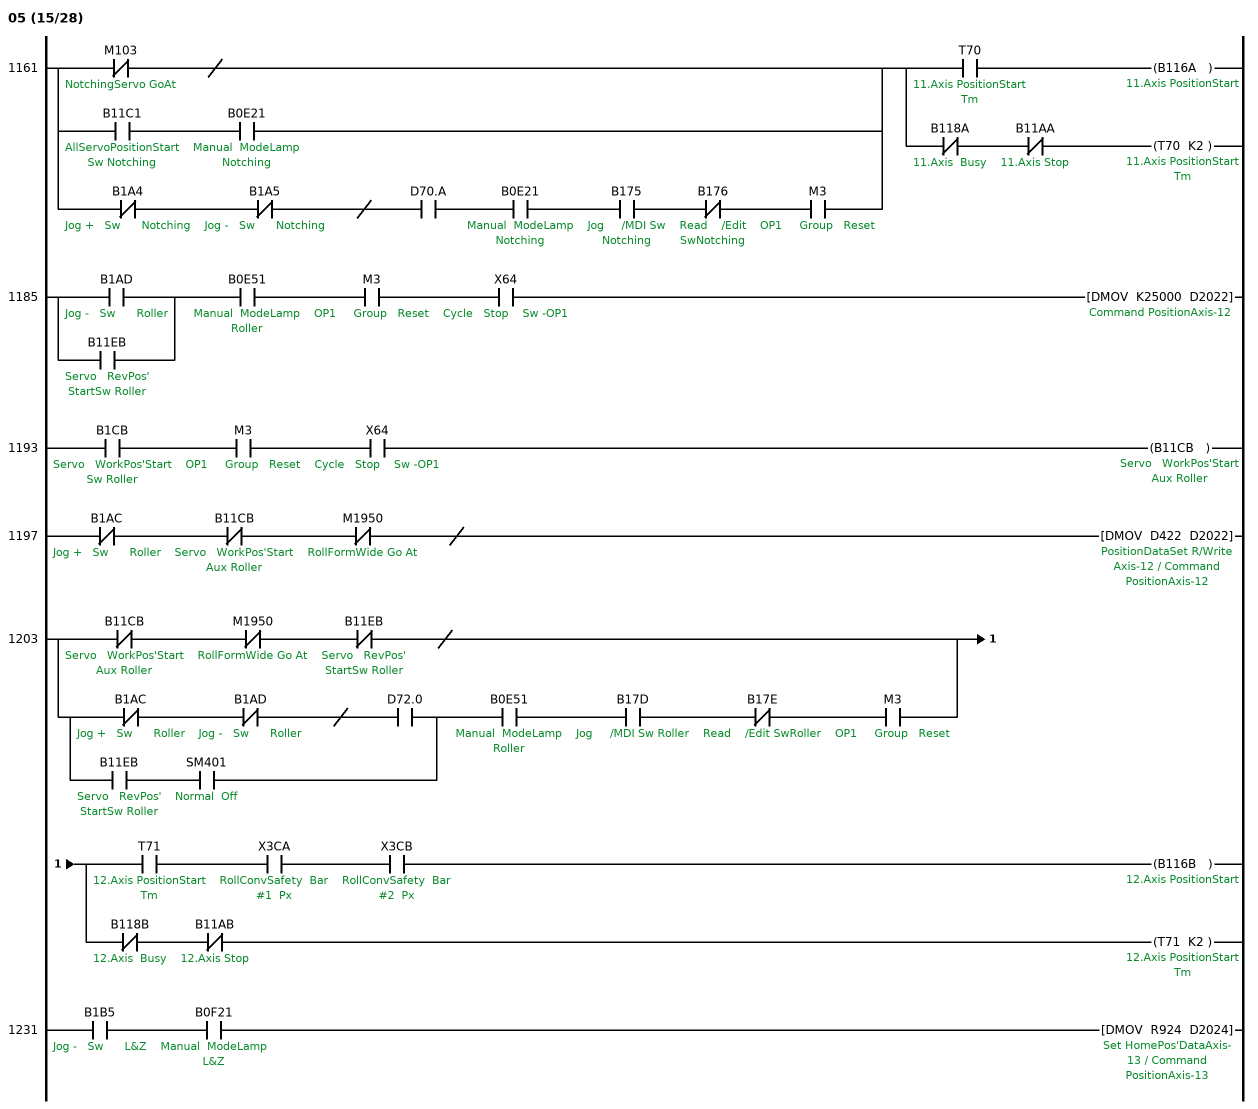
1161  LDI     M103  ; NotchingServo GoAt
      INV
      LD      B11C1  ; AllServoPositionStartSw Notching
      AND     B0E21  ; Manual  ModeLampNotching
      ORB
      LDI     B1A4  ; Jog +   Sw      Notching
      ANI     B1A5  ; Jog -   Sw      Notching
      INV
      AND     D70.A
      AND     B0E21  ; Manual  ModeLampNotching
      AND     B175  ; Jog     /MDI Sw Notching
      ANI     B176  ; Read    /Edit SwNotching
      AND     M3  ; OP1     Group   Reset
      ORB
      MPS
      AND     T70  ; 11.Axis PositionStart Tm
      OUT     B116A  ; 11.Axis PositionStart
      MPP
      ANI     B118A  ; 11.Axis  Busy
      ANI     B11AA  ; 11.Axis Stop
      OUT     T70 K2  ; 11.Axis PositionStart Tm
1185  LD      B1AD  ; Jog -   Sw      Roller
      OR      B11EB  ; Servo   RevPos' StartSw Roller
      AND     B0E51  ; Manual  ModeLampRoller
      AND     M3  ; OP1     Group   Reset
      AND     X64  ; Cycle   Stop    Sw -OP1
      DMOV    K25000 D2022  ; Command PositionAxis-12
1193  LD      B1CB  ; Servo   WorkPos'StartSw Roller
      AND     M3  ; OP1     Group   Reset
      AND     X64  ; Cycle   Stop    Sw -OP1
      OUT     B11CB  ; Servo   WorkPos'StartAux Roller
1197  LDI     B1AC  ; Jog +   Sw      Roller
      ANI     B11CB  ; Servo   WorkPos'StartAux Roller
      ANI     M1950  ; RollFormWide Go At
      INV
      DMOV    D422 D2022  ; PositionDataSet R/Write Axis-12
1203  LDI     B11CB  ; Servo   WorkPos'StartAux Roller
      ANI     M1950  ; RollFormWide Go At
      ANI     B11EB  ; Servo   RevPos' StartSw Roller
      INV
      LDI     B1AC  ; Jog +   Sw      Roller
      ANI     B1AD  ; Jog -   Sw      Roller
      INV
      AND     D72.0
      LD      B11EB  ; Servo   RevPos' StartSw Roller
      AND     SM401  ; Normal  Off
      ORB
      AND     B0E51  ; Manual  ModeLampRoller
      AND     B17D  ; Jog     /MDI Sw Roller
      ANI     B17E  ; Read    /Edit SwRoller
      AND     M3  ; OP1     Group   Reset
      ORB
      MPS
      AND     T71  ; 12.Axis PositionStart Tm
      AND     X3CA  ; RollConvSafety  Bar #1  Px
      AND     X3CB  ; RollConvSafety  Bar #2  Px
      OUT     B116B  ; 12.Axis PositionStart
      MPP
      ANI     B118B  ; 12.Axis  Busy
      ANI     B11AB  ; 12.Axis Stop
      OUT     T71 K2  ; 12.Axis PositionStart Tm
1231  LD      B1B5  ; Jog -   Sw      L&Z
      AND     B0F21  ; Manual  ModeLampL&Z
      DMOV    R924 D2024  ; Set HomePos'DataAxis-13 / Command PositionAxis-13
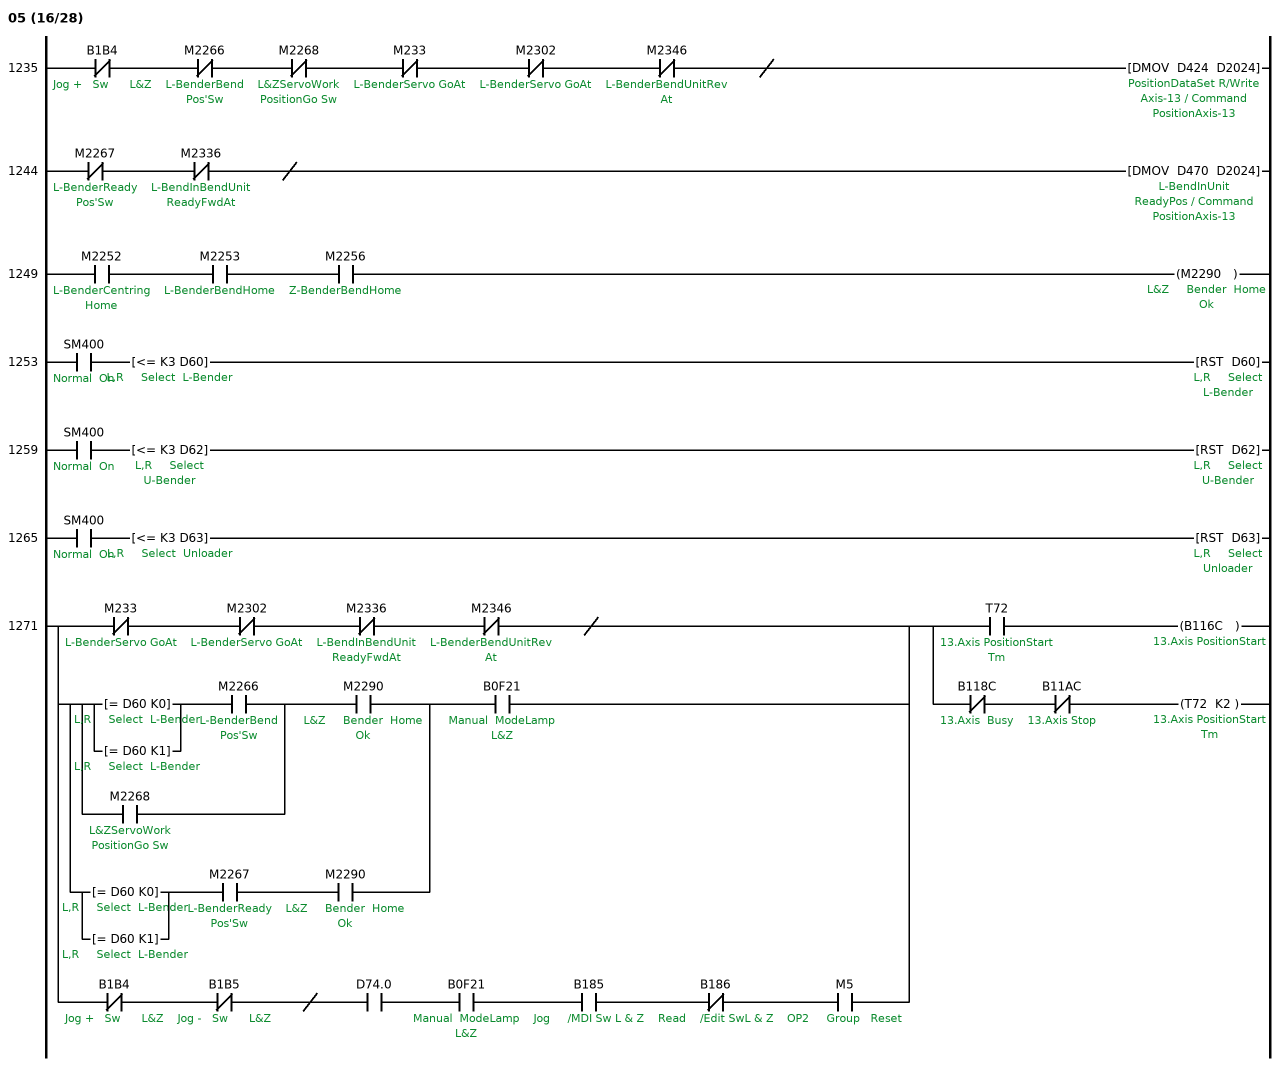
1235  LDI     B1B4  ; Jog +   Sw      L&Z
      ANI     M2266  ; L-BenderBend    Pos'Sw
      ANI     M2268  ; L&ZServoWork    PositionGo Sw
      ANI     M233  ; L-BenderServo GoAt
      ANI     M2302  ; L-BenderServo GoAt
      ANI     M2346  ; L-BenderBendUnitRev At
      INV
      DMOV    D424 D2024  ; PositionDataSet R/Write Axis-13
1244  LDI     M2267  ; L-BenderReady   Pos'Sw
      ANI     M2336  ; L-BendInBendUnitReadyFwdAt
      INV
      DMOV    D470 D2024  ; L-BendInUnit    ReadyPos
1249  LD      M2252  ; L-BenderCentringHome
      AND     M2253  ; L-BenderBendHome
      AND     M2256  ; Z-BenderBendHome
      OUT     M2290  ; L&Z     Bender  Home Ok
1253  LD      SM400  ; Normal  On
      AND<=   K3 D60  ; L,R     Select  L-Bender
      RST     D60  ; L,R     Select  L-Bender
1259  LD      SM400  ; Normal  On
      AND<=   K3 D62  ; L,R     Select  U-Bender
      RST     D62  ; L,R     Select  U-Bender
1265  LD      SM400  ; Normal  On
      AND<=   K3 D63  ; L,R     Select  Unloader
      RST     D63  ; L,R     Select  Unloader
1271  LDI     M233  ; L-BenderServo GoAt
      ANI     M2302  ; L-BenderServo GoAt
      ANI     M2336  ; L-BendInBendUnitReadyFwdAt
      ANI     M2346  ; L-BenderBendUnitRev At
      INV
      LD=     D60 K0  ; L,R     Select  L-Bender
      OR=     D60 K1  ; L,R     Select  L-Bender
      AND     M2266  ; L-BenderBend    Pos'Sw
      OR      M2268  ; L&ZServoWork    PositionGo Sw
      AND     M2290  ; L&Z     Bender  Home Ok
      LD=     D60 K0  ; L,R     Select  L-Bender
      OR=     D60 K1  ; L,R     Select  L-Bender
      AND     M2267  ; L-BenderReady   Pos'Sw
      AND     M2290  ; L&Z     Bender  Home Ok
      ORB
      AND     B0F21  ; Manual  ModeLampL&Z
      ORB
      LDI     B1B4  ; Jog +   Sw      L&Z
      ANI     B1B5  ; Jog -   Sw      L&Z
      INV
      AND     D74.0
      AND     B0F21  ; Manual  ModeLampL&Z
      AND     B185  ; Jog     /MDI Sw L & Z
      ANI     B186  ; Read    /Edit SwL & Z
      AND     M5  ; OP2     Group   Reset
      ORB
      MPS
      AND     T72  ; 13.Axis PositionStart Tm
      OUT     B116C  ; 13.Axis PositionStart
      MPP
      ANI     B118C  ; 13.Axis  Busy
      ANI     B11AC  ; 13.Axis Stop
      OUT     T72 K2  ; 13.Axis PositionStart Tm
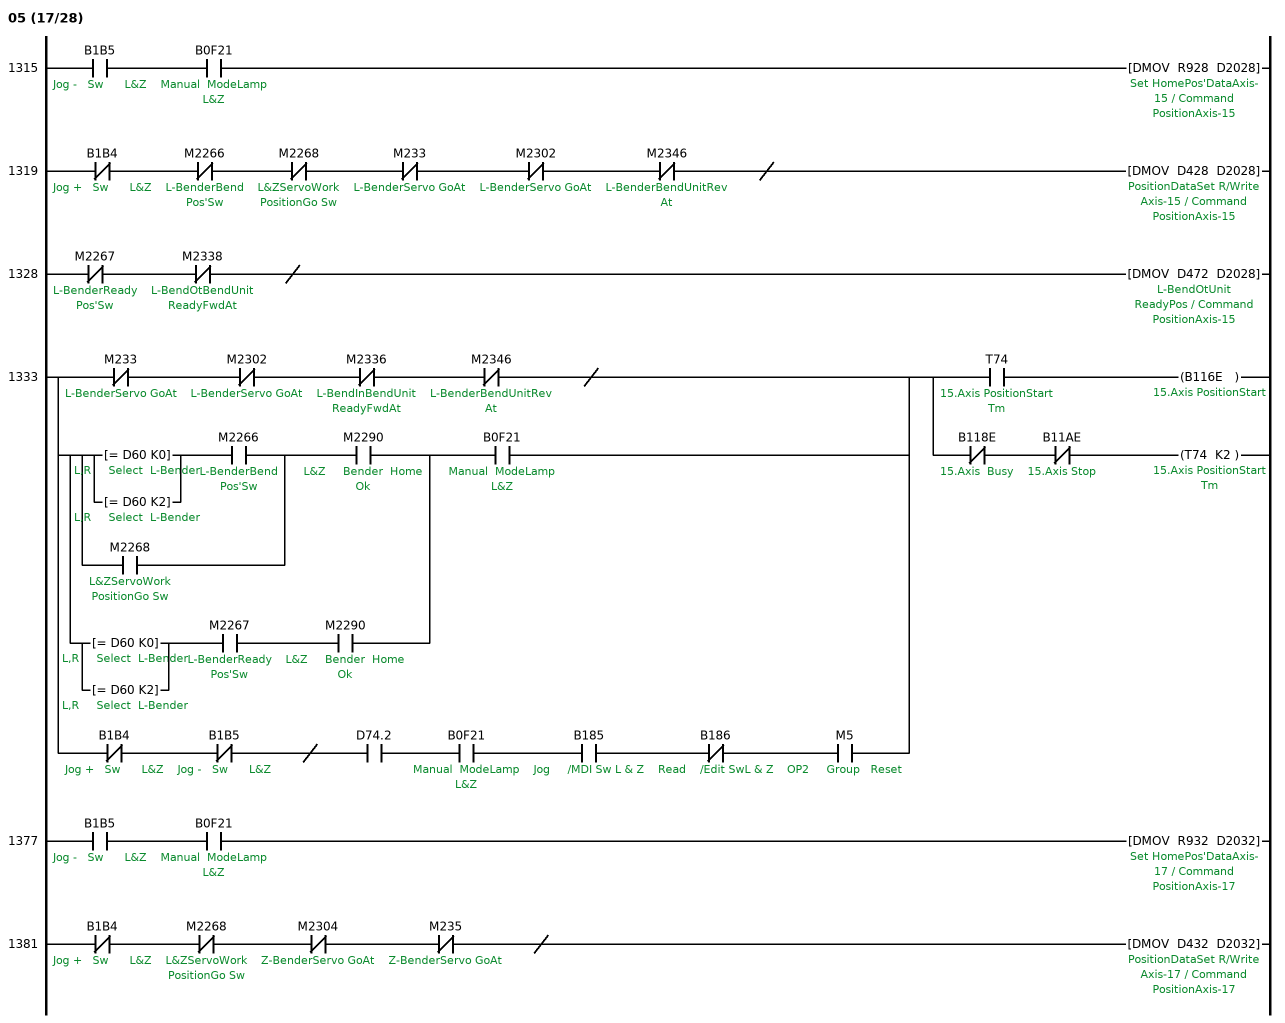
1315  LD      B1B5  ; Jog -   Sw      L&Z
      AND     B0F21  ; Manual  ModeLampL&Z
      DMOV    R928 D2028  ; Set HomePos'DataAxis-15 / Command PositionAxis-15
1319  LDI     B1B4  ; Jog +   Sw      L&Z
      ANI     M2266  ; L-BenderBend    Pos'Sw
      ANI     M2268  ; L&ZServoWork    PositionGo Sw
      ANI     M233  ; L-BenderServo GoAt
      ANI     M2302  ; L-BenderServo GoAt
      ANI     M2346  ; L-BenderBendUnitRev At
      INV
      DMOV    D428 D2028  ; PositionDataSet R/Write Axis-15
1328  LDI     M2267  ; L-BenderReady   Pos'Sw
      ANI     M2338  ; L-BendOtBendUnitReadyFwdAt
      INV
      DMOV    D472 D2028  ; L-BendOtUnit    ReadyPos
1333  LDI     M233  ; L-BenderServo GoAt
      ANI     M2302  ; L-BenderServo GoAt
      ANI     M2336  ; L-BendInBendUnitReadyFwdAt
      ANI     M2346  ; L-BenderBendUnitRev At
      INV
      LD=     D60 K0  ; L,R     Select  L-Bender
      OR=     D60 K2  ; L,R     Select  L-Bender
      AND     M2266  ; L-BenderBend    Pos'Sw
      OR      M2268  ; L&ZServoWork    PositionGo Sw
      AND     M2290  ; L&Z     Bender  Home Ok
      LD=     D60 K0  ; L,R     Select  L-Bender
      OR=     D60 K2  ; L,R     Select  L-Bender
      AND     M2267  ; L-BenderReady   Pos'Sw
      AND     M2290  ; L&Z     Bender  Home Ok
      ORB
      AND     B0F21  ; Manual  ModeLampL&Z
      ORB
      LDI     B1B4  ; Jog +   Sw      L&Z
      ANI     B1B5  ; Jog -   Sw      L&Z
      INV
      AND     D74.2
      AND     B0F21  ; Manual  ModeLampL&Z
      AND     B185  ; Jog     /MDI Sw L & Z
      ANI     B186  ; Read    /Edit SwL & Z
      AND     M5  ; OP2     Group   Reset
      ORB
      MPS
      AND     T74  ; 15.Axis PositionStart Tm
      OUT     B116E  ; 15.Axis PositionStart
      MPP
      ANI     B118E  ; 15.Axis  Busy
      ANI     B11AE  ; 15.Axis Stop
      OUT     T74 K2  ; 15.Axis PositionStart Tm
1377  LD      B1B5  ; Jog -   Sw      L&Z
      AND     B0F21  ; Manual  ModeLampL&Z
      DMOV    R932 D2032  ; Set HomePos'DataAxis-17 / Command PositionAxis-17
1381  LDI     B1B4  ; Jog +   Sw      L&Z
      ANI     M2268  ; L&ZServoWork    PositionGo Sw
      ANI     M2304  ; Z-BenderServo GoAt
      ANI     M235  ; Z-BenderServo GoAt
      INV
      DMOV    D432 D2032  ; PositionDataSet R/Write Axis-17
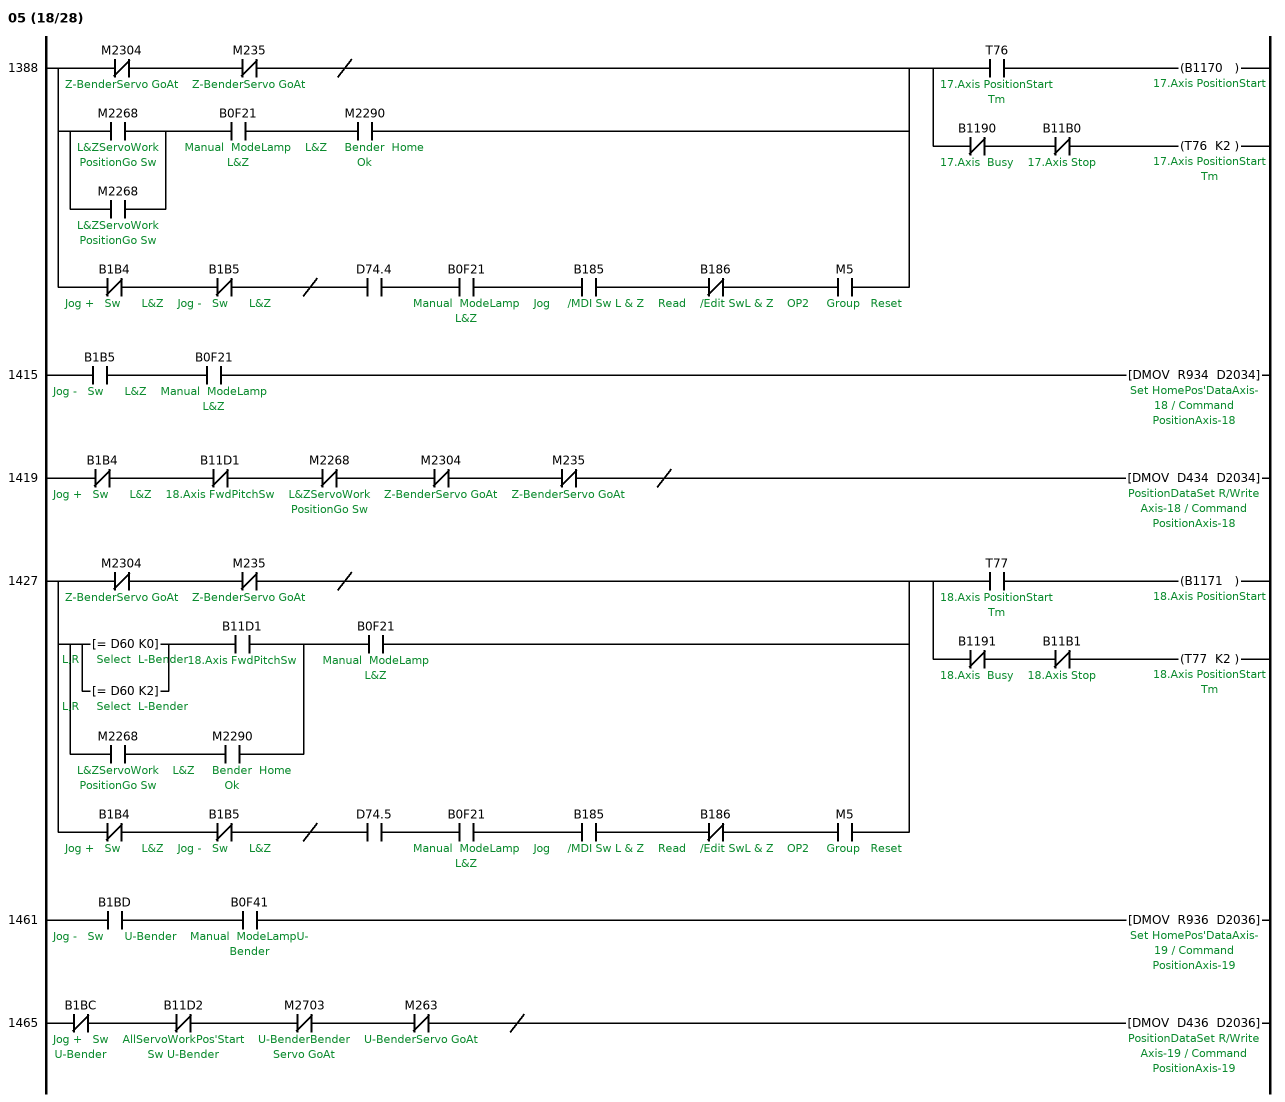
1388  LDI     M2304  ; Z-BenderServo GoAt
      ANI     M235  ; Z-BenderServo GoAt
      INV
      LD      M2268  ; L&ZServoWork    PositionGo Sw
      OR      M2268  ; L&ZServoWork    PositionGo Sw
      AND     B0F21  ; Manual  ModeLampL&Z
      AND     M2290  ; L&Z     Bender  Home Ok
      ORB
      LDI     B1B4  ; Jog +   Sw      L&Z
      ANI     B1B5  ; Jog -   Sw      L&Z
      INV
      AND     D74.4
      AND     B0F21  ; Manual  ModeLampL&Z
      AND     B185  ; Jog     /MDI Sw L & Z
      ANI     B186  ; Read    /Edit SwL & Z
      AND     M5  ; OP2     Group   Reset
      ORB
      MPS
      AND     T76  ; 17.Axis PositionStart Tm
      OUT     B1170  ; 17.Axis PositionStart
      MPP
      ANI     B1190  ; 17.Axis  Busy
      ANI     B11B0  ; 17.Axis Stop
      OUT     T76 K2  ; 17.Axis PositionStart Tm
1415  LD      B1B5  ; Jog -   Sw      L&Z
      AND     B0F21  ; Manual  ModeLampL&Z
      DMOV    R934 D2034  ; Set HomePos'DataAxis-18 / Command PositionAxis-18
1419  LDI     B1B4  ; Jog +   Sw      L&Z
      ANI     B11D1  ; 18.Axis FwdPitchSw
      ANI     M2268  ; L&ZServoWork    PositionGo Sw
      ANI     M2304  ; Z-BenderServo GoAt
      ANI     M235  ; Z-BenderServo GoAt
      INV
      DMOV    D434 D2034  ; PositionDataSet R/Write Axis-18
1427  LDI     M2304  ; Z-BenderServo GoAt
      ANI     M235  ; Z-BenderServo GoAt
      INV
      LD=     D60 K0  ; L,R     Select  L-Bender
      OR=     D60 K2  ; L,R     Select  L-Bender
      AND     B11D1  ; 18.Axis FwdPitchSw
      LD      M2268  ; L&ZServoWork    PositionGo Sw
      AND     M2290  ; L&Z     Bender  Home Ok
      ORB
      AND     B0F21  ; Manual  ModeLampL&Z
      ORB
      LDI     B1B4  ; Jog +   Sw      L&Z
      ANI     B1B5  ; Jog -   Sw      L&Z
      INV
      AND     D74.5
      AND     B0F21  ; Manual  ModeLampL&Z
      AND     B185  ; Jog     /MDI Sw L & Z
      ANI     B186  ; Read    /Edit SwL & Z
      AND     M5  ; OP2     Group   Reset
      ORB
      MPS
      AND     T77  ; 18.Axis PositionStart Tm
      OUT     B1171  ; 18.Axis PositionStart
      MPP
      ANI     B1191  ; 18.Axis  Busy
      ANI     B11B1  ; 18.Axis Stop
      OUT     T77 K2  ; 18.Axis PositionStart Tm
1461  LD      B1BD  ; Jog -   Sw      U-Bender
      AND     B0F41  ; Manual  ModeLampU-Bender
      DMOV    R936 D2036  ; Set HomePos'DataAxis-19 / Command PositionAxis-19
1465  LDI     B1BC  ; Jog +   Sw      U-Bender
      ANI     B11D2  ; AllServoWorkPos'StartSw U-Bender
      ANI     M2703  ; U-BenderBender  Servo GoAt
      ANI     M263  ; U-BenderServo GoAt
      INV
      DMOV    D436 D2036  ; PositionDataSet R/Write Axis-19
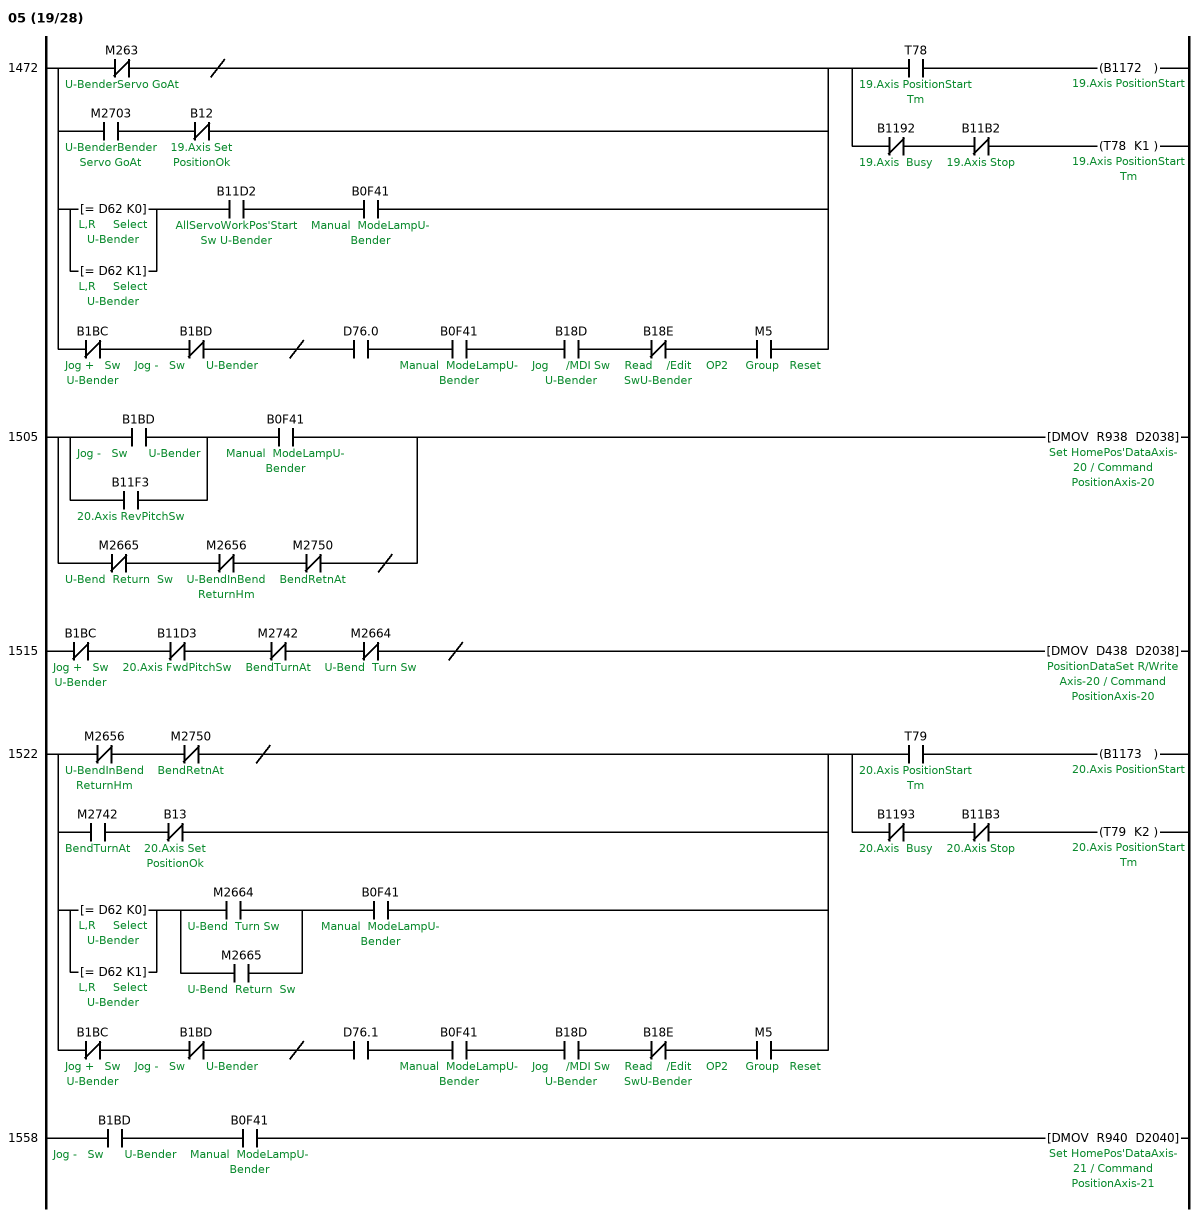
1472  LDI     M263  ; U-BenderServo GoAt
      INV
      LD      M2703  ; U-BenderBender  Servo GoAt
      ANI     B12  ; 19.Axis Set     PositionOk
      ORB
      LD=     D62 K0  ; L,R     Select  U-Bender
      OR=     D62 K1  ; L,R     Select  U-Bender
      AND     B11D2  ; AllServoWorkPos'StartSw U-Bender
      AND     B0F41  ; Manual  ModeLampU-Bender
      ORB
      LDI     B1BC  ; Jog +   Sw      U-Bender
      ANI     B1BD  ; Jog -   Sw      U-Bender
      INV
      AND     D76.0
      AND     B0F41  ; Manual  ModeLampU-Bender
      AND     B18D  ; Jog     /MDI Sw U-Bender
      ANI     B18E  ; Read    /Edit SwU-Bender
      AND     M5  ; OP2     Group   Reset
      ORB
      MPS
      AND     T78  ; 19.Axis PositionStart Tm
      OUT     B1172  ; 19.Axis PositionStart
      MPP
      ANI     B1192  ; 19.Axis  Busy
      ANI     B11B2  ; 19.Axis Stop
      OUT     T78 K1  ; 19.Axis PositionStart Tm
1505  LD      B1BD  ; Jog -   Sw      U-Bender
      OR      B11F3  ; 20.Axis RevPitchSw
      AND     B0F41  ; Manual  ModeLampU-Bender
      LDI     M2665  ; U-Bend  Return  Sw
      ANI     M2656  ; U-BendInBend    ReturnHm
      ANI     M2750  ; BendRetnAt
      INV
      ORB
      DMOV    R938 D2038  ; Set HomePos'DataAxis-20 / Command PositionAxis-20
1515  LDI     B1BC  ; Jog +   Sw      U-Bender
      ANI     B11D3  ; 20.Axis FwdPitchSw
      ANI     M2742  ; BendTurnAt
      ANI     M2664  ; U-Bend  Turn Sw
      INV
      DMOV    D438 D2038  ; PositionDataSet R/Write Axis-20
1522  LDI     M2656  ; U-BendInBend    ReturnHm
      ANI     M2750  ; BendRetnAt
      INV
      LD      M2742  ; BendTurnAt
      ANI     B13  ; 20.Axis Set     PositionOk
      ORB
      LD=     D62 K0  ; L,R     Select  U-Bender
      OR=     D62 K1  ; L,R     Select  U-Bender
      LD      M2664  ; U-Bend  Turn Sw
      OR      M2665  ; U-Bend  Return  Sw
      ANB
      AND     B0F41  ; Manual  ModeLampU-Bender
      ORB
      LDI     B1BC  ; Jog +   Sw      U-Bender
      ANI     B1BD  ; Jog -   Sw      U-Bender
      INV
      AND     D76.1
      AND     B0F41  ; Manual  ModeLampU-Bender
      AND     B18D  ; Jog     /MDI Sw U-Bender
      ANI     B18E  ; Read    /Edit SwU-Bender
      AND     M5  ; OP2     Group   Reset
      ORB
      MPS
      AND     T79  ; 20.Axis PositionStart Tm
      OUT     B1173  ; 20.Axis PositionStart
      MPP
      ANI     B1193  ; 20.Axis  Busy
      ANI     B11B3  ; 20.Axis Stop
      OUT     T79 K2  ; 20.Axis PositionStart Tm
1558  LD      B1BD  ; Jog -   Sw      U-Bender
      AND     B0F41  ; Manual  ModeLampU-Bender
      DMOV    R940 D2040  ; Set HomePos'DataAxis-21 / Command PositionAxis-21
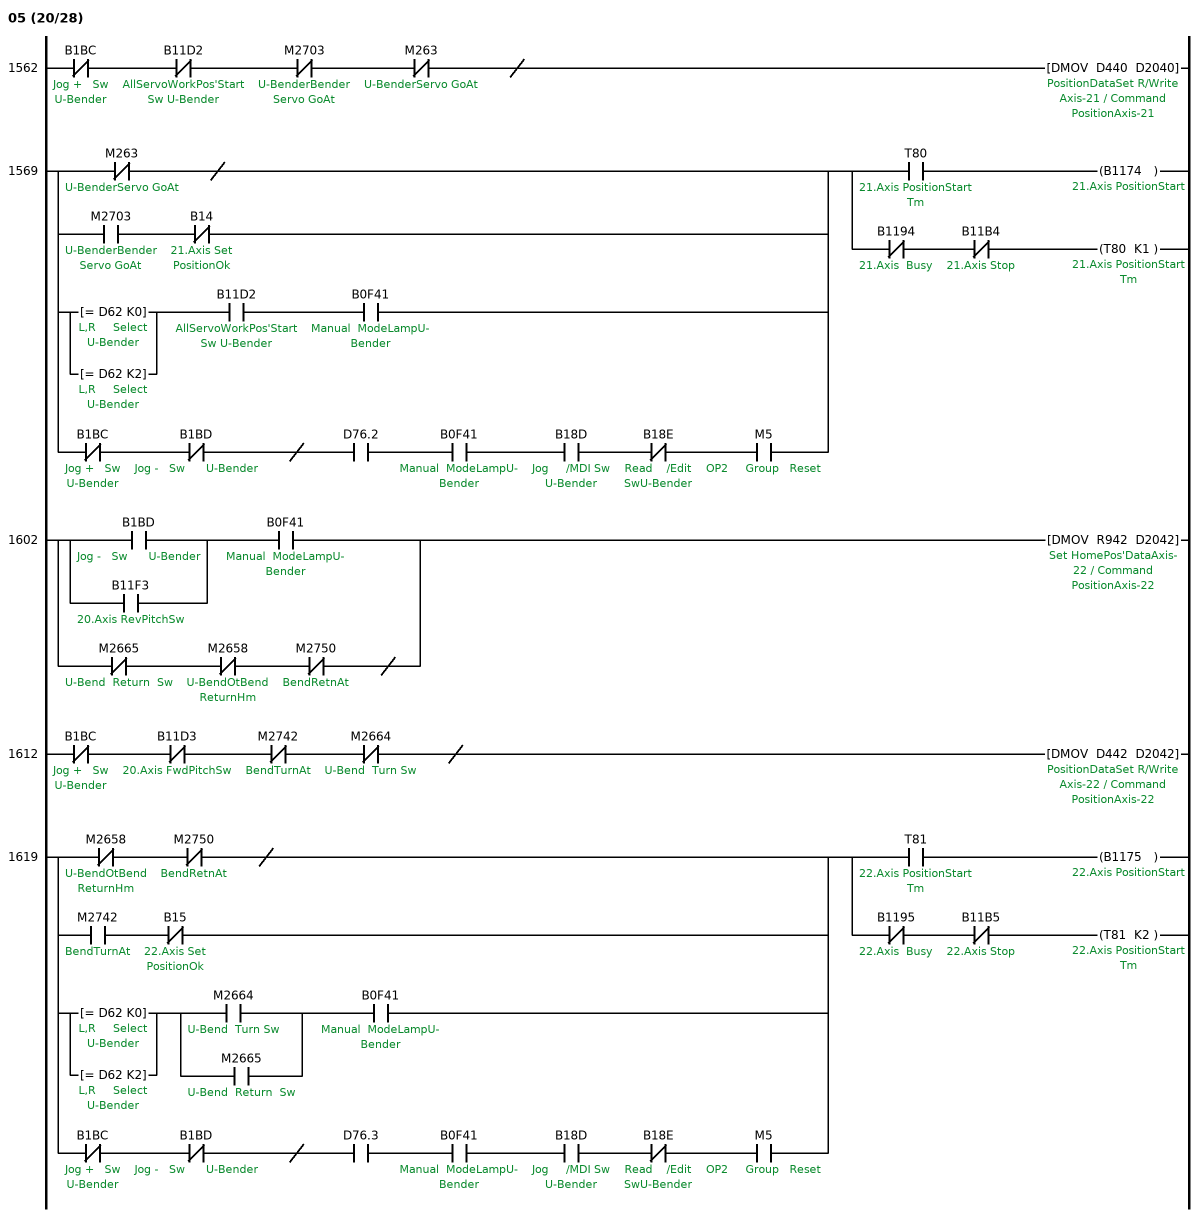
1562  LDI     B1BC  ; Jog +   Sw      U-Bender
      ANI     B11D2  ; AllServoWorkPos'StartSw U-Bender
      ANI     M2703  ; U-BenderBender  Servo GoAt
      ANI     M263  ; U-BenderServo GoAt
      INV
      DMOV    D440 D2040  ; PositionDataSet R/Write Axis-21
1569  LDI     M263  ; U-BenderServo GoAt
      INV
      LD      M2703  ; U-BenderBender  Servo GoAt
      ANI     B14  ; 21.Axis Set     PositionOk
      ORB
      LD=     D62 K0  ; L,R     Select  U-Bender
      OR=     D62 K2  ; L,R     Select  U-Bender
      AND     B11D2  ; AllServoWorkPos'StartSw U-Bender
      AND     B0F41  ; Manual  ModeLampU-Bender
      ORB
      LDI     B1BC  ; Jog +   Sw      U-Bender
      ANI     B1BD  ; Jog -   Sw      U-Bender
      INV
      AND     D76.2
      AND     B0F41  ; Manual  ModeLampU-Bender
      AND     B18D  ; Jog     /MDI Sw U-Bender
      ANI     B18E  ; Read    /Edit SwU-Bender
      AND     M5  ; OP2     Group   Reset
      ORB
      MPS
      AND     T80  ; 21.Axis PositionStart Tm
      OUT     B1174  ; 21.Axis PositionStart
      MPP
      ANI     B1194  ; 21.Axis  Busy
      ANI     B11B4  ; 21.Axis Stop
      OUT     T80 K1  ; 21.Axis PositionStart Tm
1602  LD      B1BD  ; Jog -   Sw      U-Bender
      OR      B11F3  ; 20.Axis RevPitchSw
      AND     B0F41  ; Manual  ModeLampU-Bender
      LDI     M2665  ; U-Bend  Return  Sw
      ANI     M2658  ; U-BendOtBend    ReturnHm
      ANI     M2750  ; BendRetnAt
      INV
      ORB
      DMOV    R942 D2042  ; Set HomePos'DataAxis-22 / Command PositionAxis-22
1612  LDI     B1BC  ; Jog +   Sw      U-Bender
      ANI     B11D3  ; 20.Axis FwdPitchSw
      ANI     M2742  ; BendTurnAt
      ANI     M2664  ; U-Bend  Turn Sw
      INV
      DMOV    D442 D2042  ; PositionDataSet R/Write Axis-22
1619  LDI     M2658  ; U-BendOtBend    ReturnHm
      ANI     M2750  ; BendRetnAt
      INV
      LD      M2742  ; BendTurnAt
      ANI     B15  ; 22.Axis Set     PositionOk
      ORB
      LD=     D62 K0  ; L,R     Select  U-Bender
      OR=     D62 K2  ; L,R     Select  U-Bender
      LD      M2664  ; U-Bend  Turn Sw
      OR      M2665  ; U-Bend  Return  Sw
      ANB
      AND     B0F41  ; Manual  ModeLampU-Bender
      ORB
      LDI     B1BC  ; Jog +   Sw      U-Bender
      ANI     B1BD  ; Jog -   Sw      U-Bender
      INV
      AND     D76.3
      AND     B0F41  ; Manual  ModeLampU-Bender
      AND     B18D  ; Jog     /MDI Sw U-Bender
      ANI     B18E  ; Read    /Edit SwU-Bender
      AND     M5  ; OP2     Group   Reset
      ORB
      MPS
      AND     T81  ; 22.Axis PositionStart Tm
      OUT     B1175  ; 22.Axis PositionStart
      MPP
      ANI     B1195  ; 22.Axis  Busy
      ANI     B11B5  ; 22.Axis Stop
      OUT     T81 K2  ; 22.Axis PositionStart Tm
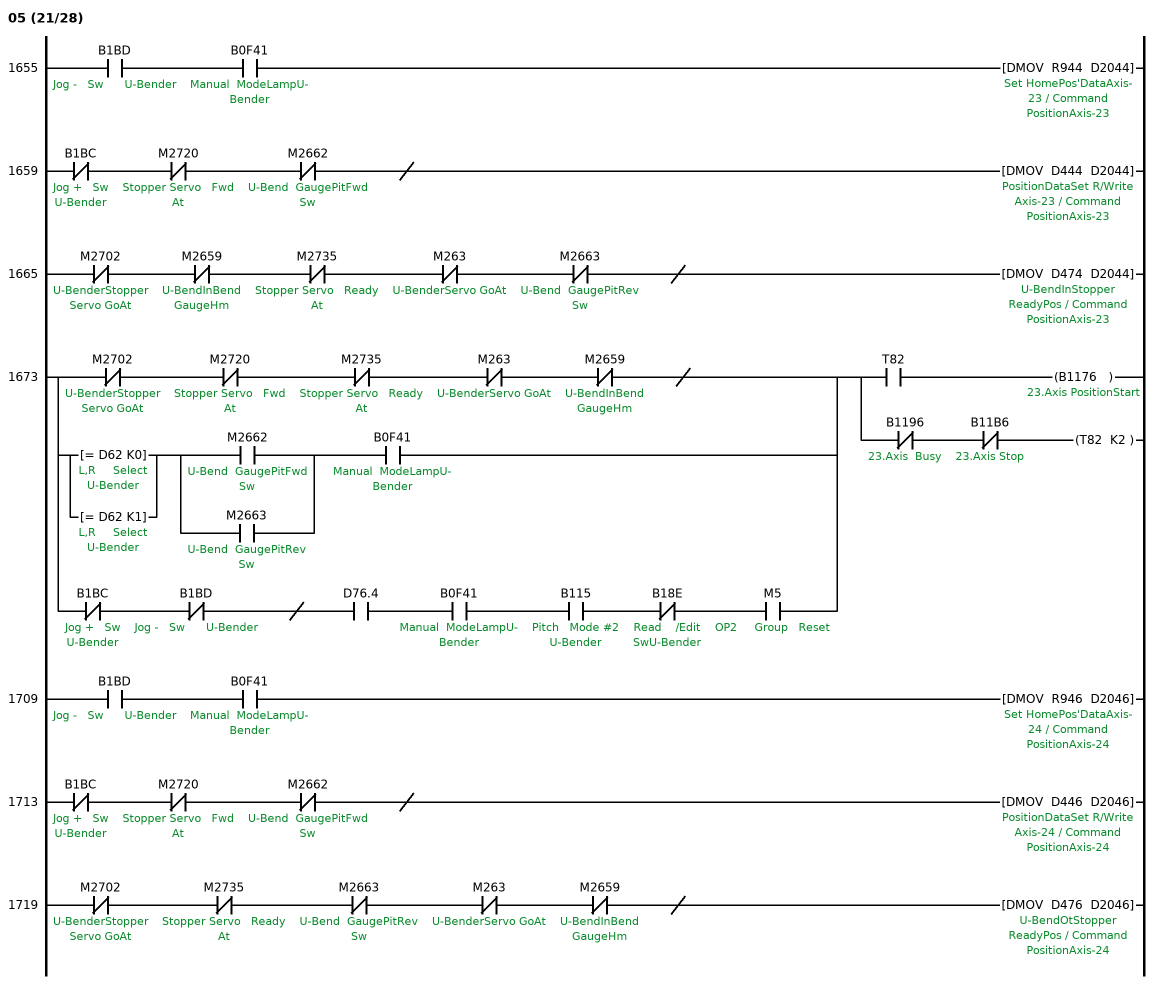
1655  LD      B1BD  ; Jog -   Sw      U-Bender
      AND     B0F41  ; Manual  ModeLampU-Bender
      DMOV    R944 D2044  ; Set HomePos'DataAxis-23 / Command PositionAxis-23
1659  LDI     B1BC  ; Jog +   Sw      U-Bender
      ANI     M2720  ; Stopper Servo   Fwd At
      ANI     M2662  ; U-Bend  GaugePitFwd Sw
      INV
      DMOV    D444 D2044  ; PositionDataSet R/Write Axis-23
1665  LDI     M2702  ; U-BenderStopper Servo GoAt
      ANI     M2659  ; U-BendInBend    GaugeHm
      ANI     M2735  ; Stopper Servo   Ready At
      ANI     M263  ; U-BenderServo GoAt
      ANI     M2663  ; U-Bend  GaugePitRev Sw
      INV
      DMOV    D474 D2044  ; U-BendInStopper ReadyPos
1673  LDI     M2702  ; U-BenderStopper Servo GoAt
      ANI     M2720  ; Stopper Servo   Fwd At
      ANI     M2735  ; Stopper Servo   Ready At
      ANI     M263  ; U-BenderServo GoAt
      ANI     M2659  ; U-BendInBend    GaugeHm
      INV
      LD=     D62 K0  ; L,R     Select  U-Bender
      OR=     D62 K1  ; L,R     Select  U-Bender
      LD      M2662  ; U-Bend  GaugePitFwd Sw
      OR      M2663  ; U-Bend  GaugePitRev Sw
      ANB
      AND     B0F41  ; Manual  ModeLampU-Bender
      ORB
      LDI     B1BC  ; Jog +   Sw      U-Bender
      ANI     B1BD  ; Jog -   Sw      U-Bender
      INV
      AND     D76.4
      AND     B0F41  ; Manual  ModeLampU-Bender
      AND     B115  ; Pitch   Mode #2 U-Bender
      ANI     B18E  ; Read    /Edit SwU-Bender
      AND     M5  ; OP2     Group   Reset
      ORB
      MPS
      AND     T82
      OUT     B1176  ; 23.Axis PositionStart
      MPP
      ANI     B1196  ; 23.Axis  Busy
      ANI     B11B6  ; 23.Axis Stop
      OUT     T82 K2
1709  LD      B1BD  ; Jog -   Sw      U-Bender
      AND     B0F41  ; Manual  ModeLampU-Bender
      DMOV    R946 D2046  ; Set HomePos'DataAxis-24 / Command PositionAxis-24
1713  LDI     B1BC  ; Jog +   Sw      U-Bender
      ANI     M2720  ; Stopper Servo   Fwd At
      ANI     M2662  ; U-Bend  GaugePitFwd Sw
      INV
      DMOV    D446 D2046  ; PositionDataSet R/Write Axis-24
1719  LDI     M2702  ; U-BenderStopper Servo GoAt
      ANI     M2735  ; Stopper Servo   Ready At
      ANI     M2663  ; U-Bend  GaugePitRev Sw
      ANI     M263  ; U-BenderServo GoAt
      ANI     M2659  ; U-BendInBend    GaugeHm
      INV
      DMOV    D476 D2046  ; U-BendOtStopper ReadyPos
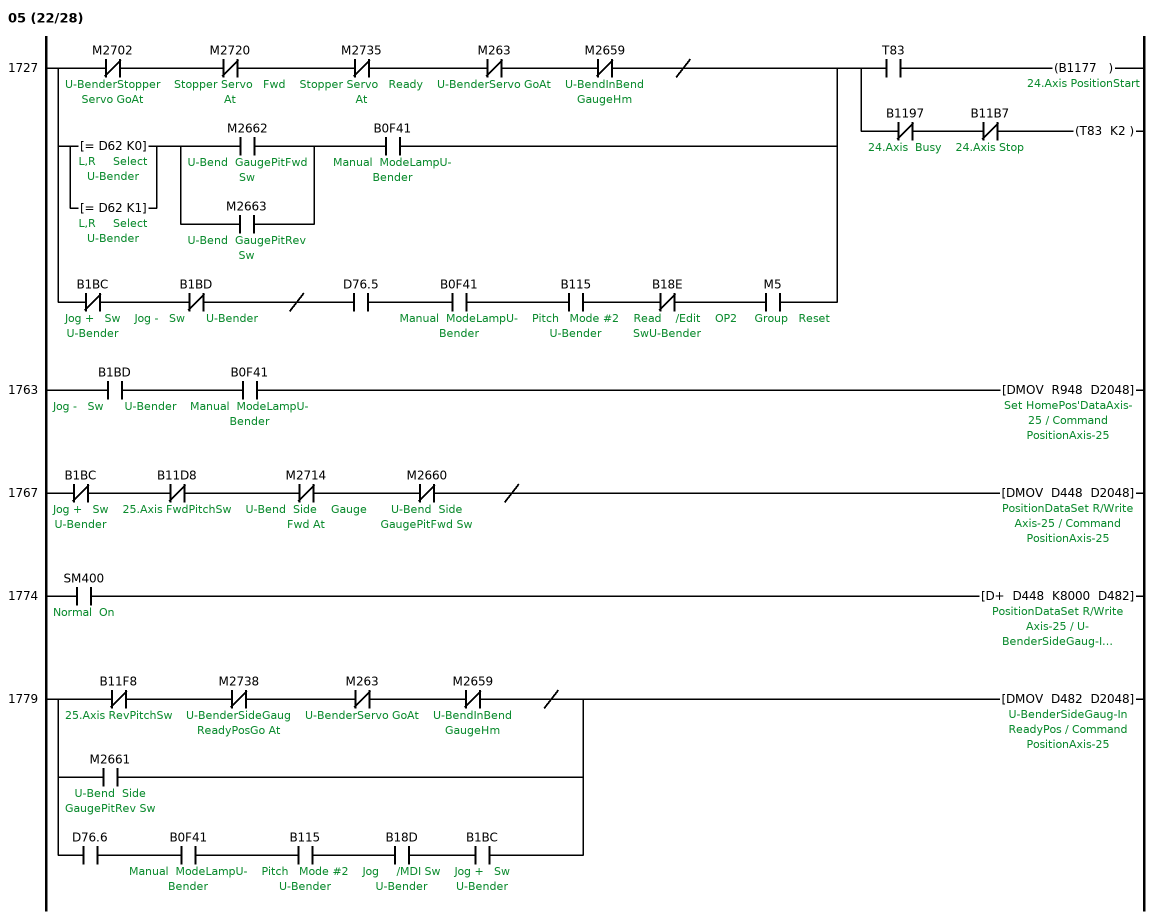
1727  LDI     M2702  ; U-BenderStopper Servo GoAt
      ANI     M2720  ; Stopper Servo   Fwd At
      ANI     M2735  ; Stopper Servo   Ready At
      ANI     M263  ; U-BenderServo GoAt
      ANI     M2659  ; U-BendInBend    GaugeHm
      INV
      LD=     D62 K0  ; L,R     Select  U-Bender
      OR=     D62 K1  ; L,R     Select  U-Bender
      LD      M2662  ; U-Bend  GaugePitFwd Sw
      OR      M2663  ; U-Bend  GaugePitRev Sw
      ANB
      AND     B0F41  ; Manual  ModeLampU-Bender
      ORB
      LDI     B1BC  ; Jog +   Sw      U-Bender
      ANI     B1BD  ; Jog -   Sw      U-Bender
      INV
      AND     D76.5
      AND     B0F41  ; Manual  ModeLampU-Bender
      AND     B115  ; Pitch   Mode #2 U-Bender
      ANI     B18E  ; Read    /Edit SwU-Bender
      AND     M5  ; OP2     Group   Reset
      ORB
      MPS
      AND     T83
      OUT     B1177  ; 24.Axis PositionStart
      MPP
      ANI     B1197  ; 24.Axis  Busy
      ANI     B11B7  ; 24.Axis Stop
      OUT     T83 K2
1763  LD      B1BD  ; Jog -   Sw      U-Bender
      AND     B0F41  ; Manual  ModeLampU-Bender
      DMOV    R948 D2048  ; Set HomePos'DataAxis-25 / Command PositionAxis-25
1767  LDI     B1BC  ; Jog +   Sw      U-Bender
      ANI     B11D8  ; 25.Axis FwdPitchSw
      ANI     M2714  ; U-Bend  Side    Gauge   Fwd At
      ANI     M2660  ; U-Bend  Side    GaugePitFwd Sw
      INV
      DMOV    D448 D2048  ; PositionDataSet R/Write Axis-25
1774  LD      SM400  ; Normal  On
      D+      D448 K8000 D482  ; U-BenderSideGaug-In     ReadyPos
1779  LDI     B11F8  ; 25.Axis RevPitchSw
      ANI     M2738  ; U-BenderSideGaugReadyPosGo At
      ANI     M263  ; U-BenderServo GoAt
      ANI     M2659  ; U-BendInBend    GaugeHm
      INV
      OR      M2661  ; U-Bend  Side    GaugePitRev Sw
      LD      D76.6
      AND     B0F41  ; Manual  ModeLampU-Bender
      AND     B115  ; Pitch   Mode #2 U-Bender
      AND     B18D  ; Jog     /MDI Sw U-Bender
      AND     B1BC  ; Jog +   Sw      U-Bender
      ORB
      DMOV    D482 D2048
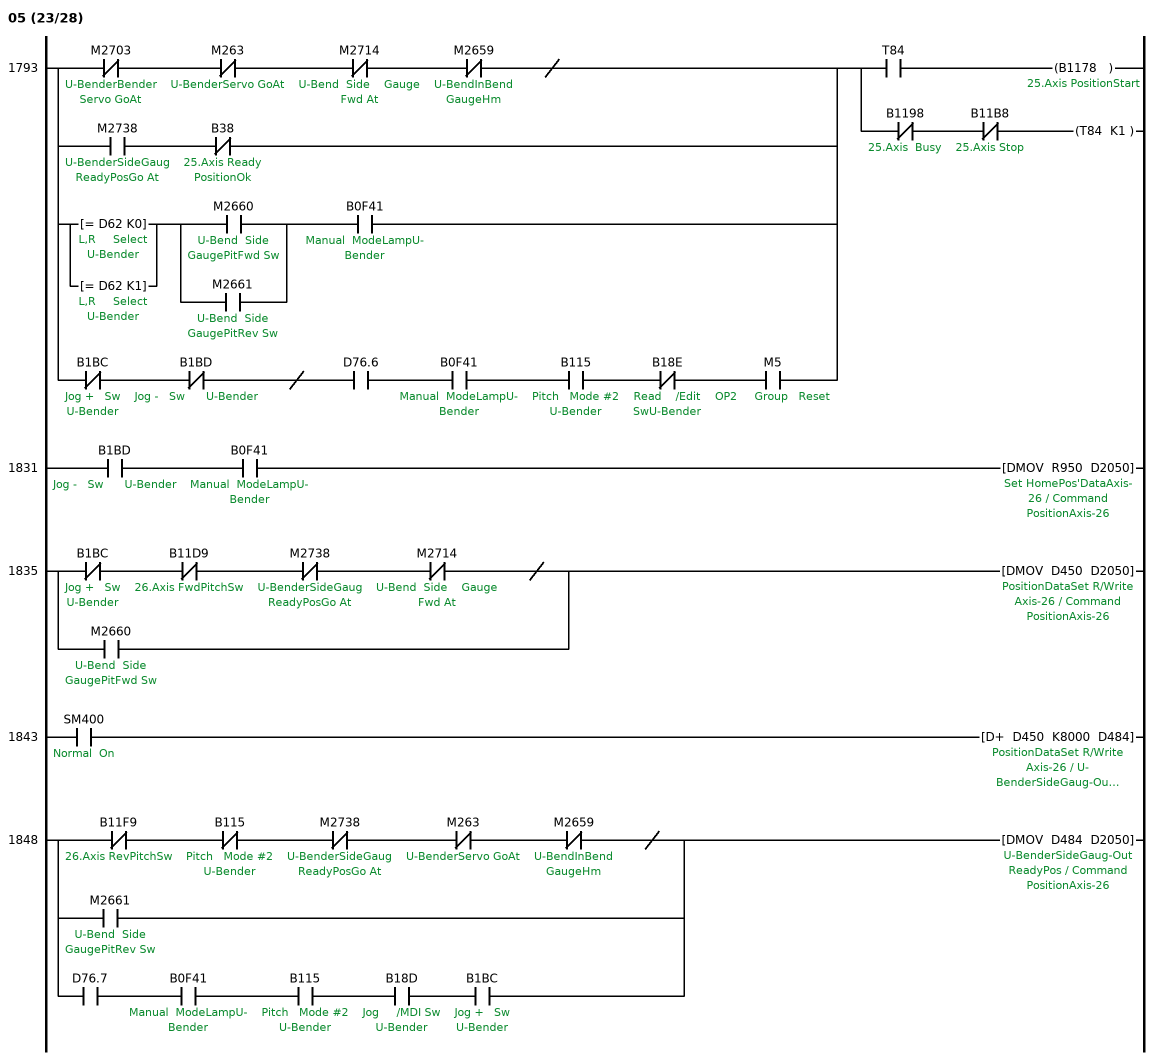
1793  LDI     M2703  ; U-BenderBender  Servo GoAt
      ANI     M263  ; U-BenderServo GoAt
      ANI     M2714  ; U-Bend  Side    Gauge   Fwd At
      ANI     M2659  ; U-BendInBend    GaugeHm
      INV
      LD      M2738  ; U-BenderSideGaugReadyPosGo At
      ANI     B38  ; 25.Axis Ready   PositionOk
      ORB
      LD=     D62 K0  ; L,R     Select  U-Bender
      OR=     D62 K1  ; L,R     Select  U-Bender
      LD      M2660  ; U-Bend  Side    GaugePitFwd Sw
      OR      M2661  ; U-Bend  Side    GaugePitRev Sw
      ANB
      AND     B0F41  ; Manual  ModeLampU-Bender
      ORB
      LDI     B1BC  ; Jog +   Sw      U-Bender
      ANI     B1BD  ; Jog -   Sw      U-Bender
      INV
      AND     D76.6
      AND     B0F41  ; Manual  ModeLampU-Bender
      AND     B115  ; Pitch   Mode #2 U-Bender
      ANI     B18E  ; Read    /Edit SwU-Bender
      AND     M5  ; OP2     Group   Reset
      ORB
      MPS
      AND     T84
      OUT     B1178  ; 25.Axis PositionStart
      MPP
      ANI     B1198  ; 25.Axis  Busy
      ANI     B11B8  ; 25.Axis Stop
      OUT     T84 K1
1831  LD      B1BD  ; Jog -   Sw      U-Bender
      AND     B0F41  ; Manual  ModeLampU-Bender
      DMOV    R950 D2050  ; Set HomePos'DataAxis-26 / Command PositionAxis-26
1835  LDI     B1BC  ; Jog +   Sw      U-Bender
      ANI     B11D9  ; 26.Axis FwdPitchSw
      ANI     M2738  ; U-BenderSideGaugReadyPosGo At
      ANI     M2714  ; U-Bend  Side    Gauge   Fwd At
      INV
      OR      M2660  ; U-Bend  Side    GaugePitFwd Sw
      DMOV    D450 D2050  ; PositionDataSet R/Write Axis-26
1843  LD      SM400  ; Normal  On
      D+      D450 K8000 D484  ; U-BenderSideGaug-Out    ReadyPos
1848  LDI     B11F9  ; 26.Axis RevPitchSw
      ANI     B115  ; Pitch   Mode #2 U-Bender
      ANI     M2738  ; U-BenderSideGaugReadyPosGo At
      ANI     M263  ; U-BenderServo GoAt
      ANI     M2659  ; U-BendInBend    GaugeHm
      INV
      OR      M2661  ; U-Bend  Side    GaugePitRev Sw
      LD      D76.7
      AND     B0F41  ; Manual  ModeLampU-Bender
      AND     B115  ; Pitch   Mode #2 U-Bender
      AND     B18D  ; Jog     /MDI Sw U-Bender
      AND     B1BC  ; Jog +   Sw      U-Bender
      ORB
      DMOV    D484 D2050
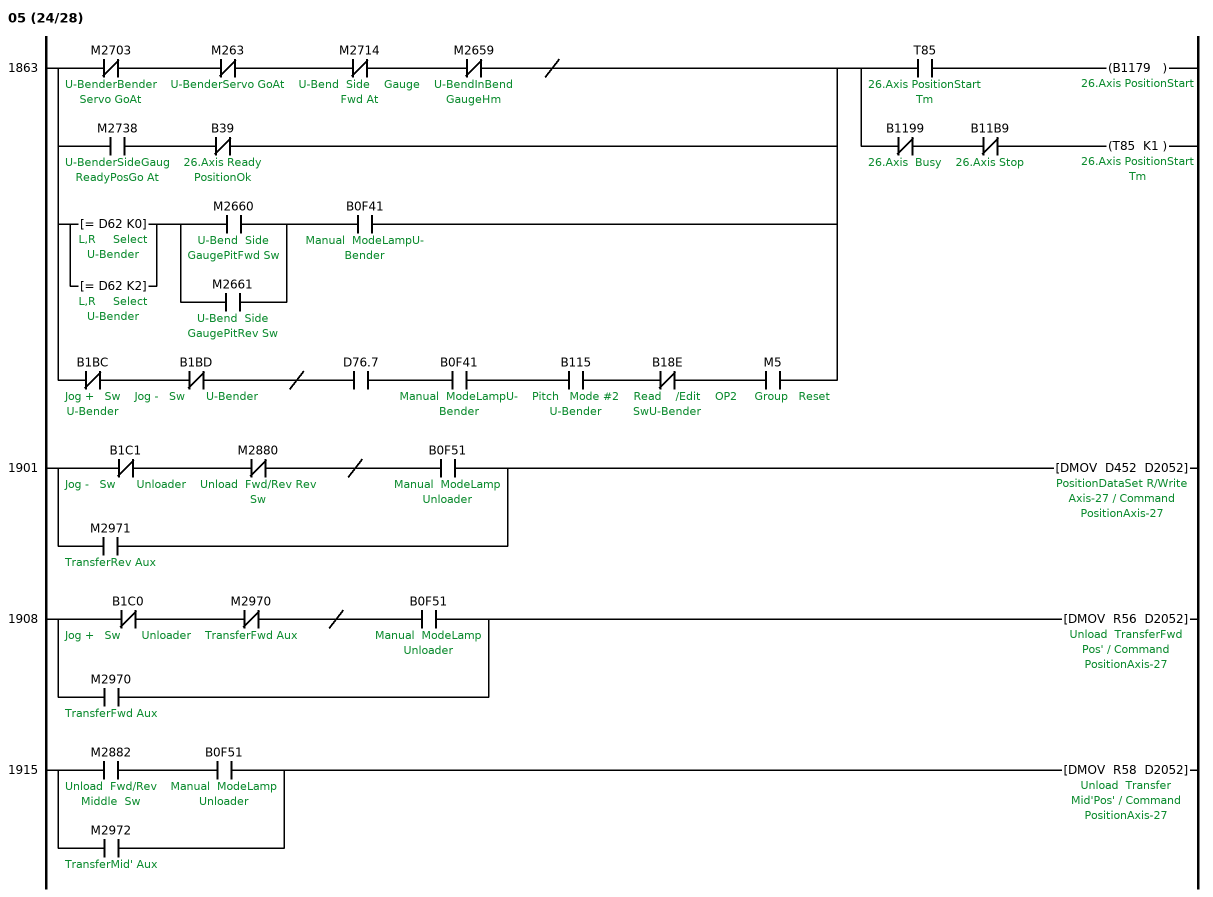
1863  LDI     M2703  ; U-BenderBender  Servo GoAt
      ANI     M263  ; U-BenderServo GoAt
      ANI     M2714  ; U-Bend  Side    Gauge   Fwd At
      ANI     M2659  ; U-BendInBend    GaugeHm
      INV
      LD      M2738  ; U-BenderSideGaugReadyPosGo At
      ANI     B39  ; 26.Axis Ready   PositionOk
      ORB
      LD=     D62 K0  ; L,R     Select  U-Bender
      OR=     D62 K2  ; L,R     Select  U-Bender
      LD      M2660  ; U-Bend  Side    GaugePitFwd Sw
      OR      M2661  ; U-Bend  Side    GaugePitRev Sw
      ANB
      AND     B0F41  ; Manual  ModeLampU-Bender
      ORB
      LDI     B1BC  ; Jog +   Sw      U-Bender
      ANI     B1BD  ; Jog -   Sw      U-Bender
      INV
      AND     D76.7
      AND     B0F41  ; Manual  ModeLampU-Bender
      AND     B115  ; Pitch   Mode #2 U-Bender
      ANI     B18E  ; Read    /Edit SwU-Bender
      AND     M5  ; OP2     Group   Reset
      ORB
      MPS
      AND     T85  ; 26.Axis PositionStart Tm
      OUT     B1179  ; 26.Axis PositionStart
      MPP
      ANI     B1199  ; 26.Axis  Busy
      ANI     B11B9  ; 26.Axis Stop
      OUT     T85 K1  ; 26.Axis PositionStart Tm
1901  LDI     B1C1  ; Jog -   Sw      Unloader
      ANI     M2880  ; Unload  Fwd/Rev Rev Sw
      INV
      AND     B0F51  ; Manual  ModeLampUnloader
      OR      M2971  ; TransferRev Aux
      DMOV    D452 D2052  ; PositionDataSet R/Write Axis-27 / Command PositionAxis-27
1908  LDI     B1C0  ; Jog +   Sw      Unloader
      ANI     M2970  ; TransferFwd Aux
      INV
      AND     B0F51  ; Manual  ModeLampUnloader
      OR      M2970  ; TransferFwd Aux
      DMOV    R56 D2052  ; Unload  TransferFwd Pos'
1915  LD      M2882  ; Unload  Fwd/Rev Middle  Sw
      AND     B0F51  ; Manual  ModeLampUnloader
      OR      M2972  ; TransferMid' Aux
      DMOV    R58 D2052  ; Unload  TransferMid'Pos'
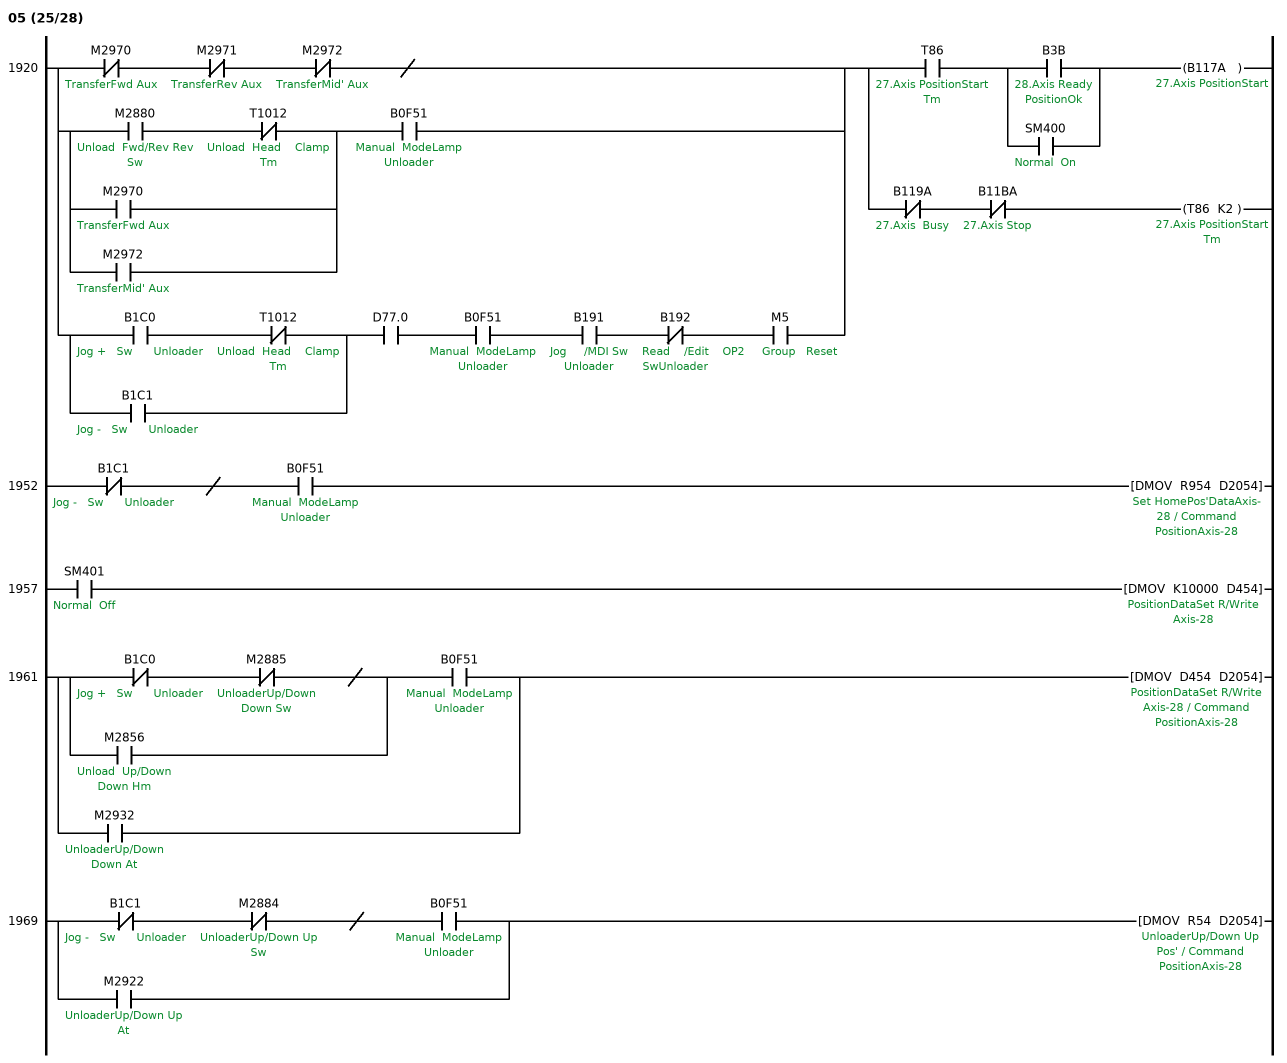
1920  LDI     M2970  ; TransferFwd Aux
      ANI     M2971  ; TransferRev Aux
      ANI     M2972  ; TransferMid' Aux
      INV
      LD      M2880  ; Unload  Fwd/Rev Rev Sw
      ANI     T1012  ; Unload  Head    Clamp Tm
      OR      M2970  ; TransferFwd Aux
      OR      M2972  ; TransferMid' Aux
      AND     B0F51  ; Manual  ModeLampUnloader
      ORB
      LD      B1C0  ; Jog +   Sw      Unloader
      ANI     T1012  ; Unload  Head    Clamp Tm
      OR      B1C1  ; Jog -   Sw      Unloader
      AND     D77.0
      AND     B0F51  ; Manual  ModeLampUnloader
      AND     B191  ; Jog     /MDI Sw Unloader
      ANI     B192  ; Read    /Edit SwUnloader
      AND     M5  ; OP2     Group   Reset
      ORB
      MPS
      AND     T86  ; 27.Axis PositionStart Tm
      LD      B3B  ; 28.Axis Ready   PositionOk
      OR      SM400  ; Normal  On
      ANB
      OUT     B117A  ; 27.Axis PositionStart
      MPP
      ANI     B119A  ; 27.Axis  Busy
      ANI     B11BA  ; 27.Axis Stop
      OUT     T86 K2  ; 27.Axis PositionStart Tm
1952  LDI     B1C1  ; Jog -   Sw      Unloader
      INV
      AND     B0F51  ; Manual  ModeLampUnloader
      DMOV    R954 D2054  ; Set HomePos'DataAxis-28 / Command PositionAxis-28
1957  LD      SM401  ; Normal  Off
      DMOV    K10000 D454  ; PositionDataSet R/Write Axis-28
1961  LDI     B1C0  ; Jog +   Sw      Unloader
      ANI     M2885  ; UnloaderUp/Down Down Sw
      INV
      OR      M2856  ; Unload  Up/Down Down Hm
      AND     B0F51  ; Manual  ModeLampUnloader
      OR      M2932  ; UnloaderUp/Down Down At
      DMOV    D454 D2054
1969  LDI     B1C1  ; Jog -   Sw      Unloader
      ANI     M2884  ; UnloaderUp/Down Up Sw
      INV
      AND     B0F51  ; Manual  ModeLampUnloader
      OR      M2922  ; UnloaderUp/Down Up At
      DMOV    R54 D2054  ; UnloaderUp/Down Up Pos'
